TEXTLIST S1_Alarms
  0 = 'Station 1 Clamp A1 Failed to Advance... Check Q1.0...' | German: 'S1 0 Row 1 Failed To Advance.. Check Qxxx.x German' | French: 'S1 0 Row 1 Failed To Advance.. Check Qxxx.x French' | 汉语: '汉语'
  1 = 'Station 1 Clamp A1 Failed to Return... Check Q1.1...' | German: 'S1 1 Row 1 Failed To Return.. Check Qxxx.x German' | French: 'S1 1 Row 1 Failed To Return.. Check Qxxx.x French' | 汉语: '汉语'
  2 = 'Station 1 Clamp A1 Lost Advanced... Check I1.0...' | German: 'S1 2 Row 1 Lost Advance Position... Check Ixxx.x German' | French: 'S1 2 Row 1 Lost Advance Position... Check Ixxx.x French' | 汉语: '汉语'
  3 = 'Station 1 Clamp A1 Lost Returned... Check I1.1...' | German: 'S1 3 Row 1 Lost Return Position... Check Ixxx.x German' | French: 'S1 3 Row 1 Lost Return Position... Check Ixxx.x French'
  4 = 'Station 1 Clamp A1 Switch Fault... Check I1.0, I1.1...' | German: 'S1 4 Row 1 Switch Fault... Check Ixxx.x / Ixxx.x German' | French: 'S1 4 Row 1 Switch Fault... Check Ixxx.x / Ixxx.x French'
  5 = 'Spare' | German: 'S1 5 Row 1 Spare Message German' | French: 'S1 5 Row 1 Spare Message French'
  6 = 'Spare' | German: 'S1 6 Row 1 Spare Message German' | French: 'S1 6 Row 1 Spare Message French'
  7 = 'Spare' | German: 'S1 7 Row 1 Spare Message German' | French: 'S1 7 Row 1 Spare Message French'
  8 = 'Spare' | German: 'S1 8 Row 1 Spare Message German' | French: 'S1 8 Row 1 Spare Message French'
  9 = 'Spare' | German: 'S1 9 Row 1 Spare Message German' | French: 'S1 9 Row 1 Spare Message French'
  10 = 'Lock Cylinder A2 Failed to Lock... Check Q1.2...' | German: 'S1 10 Row 2 Failed To Advance.. Check Qxxx.x German' | French: 'S1 10 Row 2 Failed To Advance.. Check Qxxx.x French'
  11 = 'Lock Cylinder A2 Failed to Unlock... Check Q1.3...' | German: 'S1 11 Row 2 Failed To Return.. Check Qxxx.x German' | French: 'S1 11 Row 2 Failed To Return.. Check Qxxx.x French'
  12 = 'Lock Cylinder A2 Lost Locked... Check I1.2...' | German: 'S1 12 Row 2 Lost Advance Position... Check Ixxx.x German' | French: 'S1 12 Row 2 Lost Advance Position... Check Ixxx.x French'
  13 = 'Lock Cylinder A2 Lost Unlocked... Check I1.3...' | German: 'S1 13 Row 2 Lost Return Position... Check Ixxx.x German' | French: 'S1 13 Row 2 Lost Return Position... Check Ixxx.x French'
  14 = 'Lock Cylinder A2 Switch Fault... Check I1.2, I1.3...' | German: 'S1 14 Row 2 Switch Fault... Check Ixxx.x / Ixxx.x German' | French: 'S1 14 Row 2 Switch Fault... Check Ixxx.x / Ixxx.x French'
  15 = 'Spare' | German: 'S1 15 Row 2 Spare Message German' | French: 'S1 15 Row 2 Spare Message French'
  16 = 'Spare' | German: 'S1 16 Row 2 Spare Message German' | French: 'S1 16 Row 2 Spare Message French'
  17 = 'Spare' | German: 'S1 17 Row 2 Spare Message German' | French: 'S1 17 Row 2 Spare Message French'
  18 = 'Spare' | German: 'S1 18 Row 2 Spare Message German' | French: 'S1 18 Row 2 Spare Message French'
  19 = 'Spare' | German: 'S1 19 Row 2 Spare Message German' | French: 'S1 19 Row 2 Spare Message French'
  20 = 'Urger Cylinder A3 Failed to Urge... Check Q1.4...' | German: 'S1 20 Row 3 Failed To Advance.. Check Qxxx.x German' | French: 'S1 20 Row 3 Failed To Advance.. Check Qxxx.x French'
  21 = 'Urger Cylinder A3 Failed to Return... Check Q1.5...' | German: 'S1 21 Row 3 Failed To Return.. Check Qxxx.x German' | French: 'S1 21 Row 3 Failed To Return.. Check Qxxx.x French'
  22 = 'Urger Cylinder A3 Lost Urged... Check I1.4...' | German: 'S1 22 Row 3 Lost Advance Position... Check Ixxx.x German' | French: 'S1 22 Row 3 Lost Advance Position... Check Ixxx.x French'
  23 = 'Urger Cylinder A3 Lost Returned... Check I1.5...' | German: 'S1 23 Row 3 Lost Return Position... Check Ixxx.x German' | French: 'S1 23 Row 3 Lost Return Position... Check Ixxx.x French'
  24 = 'Urger Cylinder A3 Switch Fault... Check I1.4, I1.5...' | German: 'S1 24 Row 3 Switch Fault... Check Ixxx.x / Ixxx.x German' | French: 'S1 24 Row 3 Switch Fault... Check Ixxx.x / Ixxx.x French'
  25 = 'Spare' | German: 'S1 25 Row 3 Spare Message German' | French: 'S1 25 Row 3 Spare Message French'
  26 = 'Spare' | German: 'S1 26 Row 3 Spare Message German' | French: 'S1 26 Row 3 Spare Message French'
  27 = 'Spare' | German: 'S1 27 Row 3 Spare Message German' | French: 'S1 27 Row 3 Spare Message French'
  28 = 'Spare' | German: 'S1 28 Row 3 Spare Message German' | French: 'S1 28 Row 3 Spare Message French'
  29 = 'Spare' | German: 'S1 29 Row 3 Spare Message German' | French: 'S1 29 Row 3 Spare Message French'
  30 = 'Clamp Cylinder A1 Failed to Advance... Check Q1.0...' | German: 'S1 30 Row 4 Failed To Advance.. Check Qxxx.x German' | French: 'S1 30 Row 4 Failed To Advance.. Check Qxxx.x French'
  31 = 'Clamp Cylinder A1 Failed to Return... Check Q1.1...' | German: 'S1 31 Row 4 Failed To Return.. Check Qxxx.x German' | French: 'S1 31 Row 4 Failed To Return.. Check Qxxx.x French'
  32 = 'Clamp Cylinder A1 Lost Advanced... Check I1.0...' | German: 'S1 32 Row 4 Lost Advance Position... Check Ixxx.x German' | French: 'S1 32 Row 4 Lost Advance Position... Check Ixxx.x French'
  33 = 'Clamp Cylinder A1 Lost Returned... Check I1.1...' | German: 'S1 33 Row 4 Lost Return Position... Check Ixxx.x German' | French: 'S1 33 Row 4 Lost Return Position... Check Ixxx.x French'
  34 = 'Clamp Cylinder A1 Switch Fault... Check I1.0, I1.1...' | German: 'S1 34 Row 4 Switch Fault... Check Ixxx.x / Ixxx.x German' | French: 'S1 34 Row 4 Switch Fault... Check Ixxx.x / Ixxx.x French'
  35 = 'Spare' | German: 'S1 35 Row 4 Spare Message German' | French: 'S1 35 Row 4 Spare Message French'
  36 = 'Spare' | German: 'S1 36 Row 4 Spare Message German' | French: 'S1 36 Row 4 Spare Message French'
  37 = 'Spare' | German: 'S1 37 Row 4 Spare Message German' | French: 'S1 37 Row 4 Spare Message French'
  38 = 'Spare' | German: 'S1 38 Row 4 Spare Message German' | French: 'S1 38 Row 4 Spare Message French'
  39 = 'Spare' | German: 'S1 39 Row 4 Spare Message German' | French: 'S1 39 Row 4 Spare Message French'
  40 = 'Clamp Cylinder A1 Failed to Advance... Check Q1.0...' | German: 'S1 40 Row 5 Failed To Advance.. Check Qxxx.x German' | French: 'S1 40 Row 5 Failed To Advance.. Check Qxxx.x French'
  41 = 'Clamp Cylinder A1 Failed to Return... Check Q1.1...' | German: 'S1 41 Row 5 Failed To Return.. Check Qxxx.x German' | French: 'S1 41 Row 5 Failed To Return.. Check Qxxx.x French'
  42 = 'Clamp Cylinder A1 Lost Advanced... Check I1.0...' | German: 'S1 42 Row 5 Lost Advance Position... Check Ixxx.x German' | French: 'S1 42 Row 5 Lost Advance Position... Check Ixxx.x French'
  43 = 'Clamp Cylinder A1 Lost Returned... Check I1.1...' | German: 'S1 43 Row 5 Lost Return Position... Check Ixxx.x German' | French: 'S1 43 Row 5 Lost Return Position... Check Ixxx.x French'
  44 = 'Clamp Cylinder A1 Switch Fault... Check I1.0, I1.1...' | German: 'S1 44 Row 5 Switch Fault... Check Ixxx.x / Ixxx.x German' | French: 'S1 44 Row 5 Switch Fault... Check Ixxx.x / Ixxx.x French'
  45 = 'Spare' | German: 'S1 45 Row 5 Spare Message German' | French: 'S1 45 Row 5 Spare Message French'
  46 = 'Spare' | German: 'S1 46 Row 5 Spare Message German' | French: 'S1 46 Row 5 Spare Message French'
  47 = 'Spare' | German: 'S1 47 Row 5 Spare Message German' | French: 'S1 47 Row 5 Spare Message French'
  48 = 'Spare' | German: 'S1 48 Row 5 Spare Message German' | French: 'S1 48 Row 5 Spare Message French'
  49 = 'Spare' | German: 'S1 49 Row 5 Spare Message German' | French: 'S1 49 Row 5 Spare Message French'
  50 = 'Clamp Cylinder A1 Failed to Advance... Check Q1.0...' | German: 'S1 50 Row 6 Failed To Advance.. Check Qxxx.x German' | French: 'S1 50 Row 6 Failed To Advance.. Check Qxxx.x French'
  51 = 'Clamp Cylinder A1 Failed to Return... Check Q1.1...' | German: 'S1 51 Row 6 Failed To Return.. Check Qxxx.x German' | French: 'S1 51 Row 6 Failed To Return.. Check Qxxx.x French'
  52 = 'Clamp Cylinder A1 Lost Advanced... Check I1.0...' | German: 'S1 52 Row 6 Lost Advance Position... Check Ixxx.x German' | French: 'S1 52 Row 6 Lost Advance Position... Check Ixxx.x French'
  53 = 'Clamp Cylinder A1 Lost Returned... Check I1.1...' | German: 'S1 53 Row 6 Lost Return Position... Check Ixxx.x German' | French: 'S1 53 Row 6 Lost Return Position... Check Ixxx.x French'
  54 = 'Clamp Cylinder A1 Switch Fault... Check I1.0, I1.1...' | German: 'S1 54 Row 6 Switch Fault... Check Ixxx.x / Ixxx.x German' | French: 'S1 54 Row 6 Switch Fault... Check Ixxx.x / Ixxx.x French'
  55 = 'Spare' | German: 'S1 55 Row 6 Spare Message German' | French: 'S1 55 Row 6 Spare Message French'
  56 = 'Spare' | German: 'S1 56 Row 6 Spare Message German' | French: 'S1 56 Row 6 Spare Message French'
  57 = 'Spare' | German: 'S1 57 Row 6 Spare Message German' | French: 'S1 57 Row 6 Spare Message French'
  58 = 'Spare' | German: 'S1 58 Row 6 Spare Message German' | French: 'S1 58 Row 6 Spare Message French'
  59 = 'Spare' | German: 'S1 59 Row 6 Spare Message German' | French: 'S1 59 Row 6 Spare Message French'
  60 = 'Clamp Cylinder A1 Failed to Advance... Check Q1.0...' | German: 'S1 60 Row 7 Failed To Advance.. Check Qxxx.x German' | French: 'S1 60 Row 7 Failed To Advance.. Check Qxxx.x French'
  61 = 'Clamp Cylinder A1 Failed to Return... Check Q1.1...' | German: 'S1 61 Row 7 Failed To Return.. Check Qxxx.x German' | French: 'S1 61 Row 7 Failed To Return.. Check Qxxx.x French'
  62 = 'Clamp Cylinder A1 Lost Advanced... Check I1.0...' | German: 'S1 62 Row 7 Lost Advance Position... Check Ixxx.x German' | French: 'S1 62 Row 7 Lost Advance Position... Check Ixxx.x French'
  63 = 'Clamp Cylinder A1 Lost Returned... Check I1.1...' | German: 'S1 63 Row 7 Lost Return Position... Check Ixxx.x German' | French: 'S1 63 Row 7 Lost Return Position... Check Ixxx.x French'
  64 = 'Clamp Cylinder A1 Switch Fault... Check I1.0, I1.1...' | German: 'S1 64 Row 7 Switch Fault... Check Ixxx.x / Ixxx.x German' | French: 'S1 64 Row 7 Switch Fault... Check Ixxx.x / Ixxx.x French'
  65 = 'Spare' | German: 'S1 65 Row 7 Spare Message German' | French: 'S1 65 Row 7 Spare Message French'
  66 = 'Spare' | German: 'S1 66 Row 7 Spare Message German' | French: 'S1 66 Row 7 Spare Message French'
  67 = 'Spare' | German: 'S1 67 Row 7 Spare Message German' | French: 'S1 67 Row 7 Spare Message French'
  68 = 'Spare' | German: 'S1 68 Row 7 Spare Message German' | French: 'S1 68 Row 7 Spare Message French'
  69 = 'Spare' | German: 'S1 69 Row 7 Spare Message German' | French: 'S1 69 Row 7 Spare Message French'
  70 = 'Clamp Cylinder A1 Failed to Advance... Check Q1.0...' | German: 'S1 70 Row 8 Failed To Advance.. Check Qxxx.x German' | French: 'S1 70 Row 8 Failed To Advance.. Check Qxxx.x French'
  71 = 'Clamp Cylinder A1 Failed to Return... Check Q1.1...' | German: 'S1 71 Row 8 Failed To Return.. Check Qxxx.x German' | French: 'S1 71 Row 8 Failed To Return.. Check Qxxx.x French'
  72 = 'Clamp Cylinder A1 Lost Advanced... Check I1.0...' | German: 'S1 72 Row 8 Lost Advance Position... Check Ixxx.x German' | French: 'S1 72 Row 8 Lost Advance Position... Check Ixxx.x French'
  73 = 'Clamp Cylinder A1 Lost Returned... Check I1.1...' | German: 'S1 73 Row 8 Lost Return Position... Check Ixxx.x German' | French: 'S1 73 Row 8 Lost Return Position... Check Ixxx.x French'
  74 = 'Clamp Cylinder A1 Switch Fault... Check I1.0, I1.1...' | German: 'S1 74 Row 8 Switch Fault... Check Ixxx.x / Ixxx.x German' | French: 'S1 74 Row 8 Switch Fault... Check Ixxx.x / Ixxx.x French'
  75 = 'Spare' | German: 'S1 75 Row 8 Spare Message German' | French: 'S1 75 Row 8 Spare Message French'
  76 = 'Spare' | German: 'S1 76 Row 8 Spare Message German' | French: 'S1 76 Row 8 Spare Message French'
  77 = 'Spare' | German: 'S1 77 Row 8 Spare Message German' | French: 'S1 77 Row 8 Spare Message French'
  78 = 'Spare' | German: 'S1 78 Row 8 Spare Message German' | French: 'S1 78 Row 8 Spare Message French'
  79 = 'Spare' | German: 'S1 79 Row 8 Spare Message German' | French: 'S1 79 Row 8 Spare Message French'
  80 = 'Clamp Cylinder A1 Failed to Advance... Check Q1.0...' | German: 'S1 80 Row 9 Failed To Advance.. Check Qxxx.x German' | French: 'S1 80 Row 9 Failed To Advance.. Check Qxxx.x French'
  81 = 'Clamp Cylinder A1 Failed to Return... Check Q1.1...' | German: 'S1 81 Row 9 Failed To Return.. Check Qxxx.x German' | French: 'S1 81 Row 9 Failed To Return.. Check Qxxx.x French'
  82 = 'Clamp Cylinder A1 Lost Advanced... Check I1.0...' | German: 'S1 82 Row 9 Lost Advance Position... Check Ixxx.x German' | French: 'S1 82 Row 9 Lost Advance Position... Check Ixxx.x French'
  83 = 'Clamp Cylinder A1 Lost Returned... Check I1.1...' | German: 'S1 83 Row 9 Lost Return Position... Check Ixxx.x German' | French: 'S1 83 Row 9 Lost Return Position... Check Ixxx.x French'
  84 = 'Clamp Cylinder A1 Switch Fault... Check I1.0, I1.1...' | German: 'S1 84 Row 9 Switch Fault... Check Ixxx.x / Ixxx.x German' | French: 'S1 84 Row 9 Switch Fault... Check Ixxx.x / Ixxx.x French'
  85 = 'Spare' | German: 'S1 85 Row 9 Spare Message German' | French: 'S1 85 Row 9 Spare Message French'
  86 = 'Spare' | German: 'S1 86 Row 9 Spare Message German' | French: 'S1 86 Row 9 Spare Message French'
  87 = 'Spare' | German: 'S1 87 Row 9 Spare Message German' | French: 'S1 87 Row 9 Spare Message French'
  88 = 'Spare' | German: 'S1 88 Row 9 Spare Message German' | French: 'S1 88 Row 9 Spare Message French'
  89 = 'Spare' | German: 'S1 89 Row 9 Spare Message German' | French: 'S1 89 Row 9 Spare Message French'
  90 = 'Clamp Cylinder A1 Failed to Advance... Check Q1.0...' | German: 'S1 90 Row 10 Failed To Advance.. Check Qxxx.x German' | French: 'S1 90 Row 10 Failed To Advance.. Check Qxxx.x French'
  91 = 'Clamp Cylinder A1 Failed to Return... Check Q1.1...' | German: 'S1 91 Row 10 Failed To Return.. Check Qxxx.x German' | French: 'S1 91 Row 10 Failed To Return.. Check Qxxx.x French'
  92 = 'Clamp Cylinder A1 Lost Advanced... Check I1.0...' | German: 'S1 92 Row 10 Lost Advance Position... Check Ixxx.x German' | French: 'S1 92 Row 10 Lost Advance Position... Check Ixxx.x French'
  93 = 'Clamp Cylinder A1 Lost Returned... Check I1.1...' | German: 'S1 93 Row 10 Lost Return Position... Check Ixxx.x German' | French: 'S1 93 Row 10 Lost Return Position... Check Ixxx.x French'
  94 = 'Clamp Cylinder A1 Switch Fault... Check I1.0, I1.1...' | German: 'S1 94 Row 10 Switch Fault... Check Ixxx.x / Ixxx.x German' | French: 'S1 94 Row 10 Switch Fault... Check Ixxx.x / Ixxx.x French'
  95 = 'Spare' | German: 'S1 95 Row 10 Spare Message German' | French: 'S1 95 Row 10 Spare Message French'
  96 = 'Spare' | German: 'S1 96 Row 10 Spare Message German' | French: 'S1 96 Row 10 Spare Message French'
  97 = 'Spare' | German: 'S1 97 Row 10 Spare Message German' | French: 'S1 97 Row 10 Spare Message French'
  98 = 'Spare' | German: 'S1 98 Row 10 Spare Message German' | French: 'S1 98 Row 10 Spare Message French'
  99 = 'Spare' | German: 'S1 99 Row 10 Spare Message German' | French: 'S1 99 Row 10 Spare Message French'
  100 = 'Clamp Cylinder A1 Failed to Advance... Check Q1.0...' | German: 'S1 100 Row 11 Failed To Advance.. Check Qxxx.x German' | French: 'S1 100 Row 11 Failed To Advance.. Check Qxxx.x French'
  101 = 'Clamp Cylinder A1 Failed to Return... Check Q1.1...' | German: 'S1 101 Row 11 Failed To Return.. Check Qxxx.x German' | French: 'S1 101 Row 11 Failed To Return.. Check Qxxx.x French'
  102 = 'Clamp Cylinder A1 Lost Advanced... Check I1.0...' | German: 'S1 102 Row 11 Lost Advance Position... Check Ixxx.x German' | French: 'S1 102 Row 11 Lost Advance Position... Check Ixxx.x French'
  103 = 'Clamp Cylinder A1 Lost Returned... Check I1.1...' | German: 'S1 103 Row 11 Lost Return Position... Check Ixxx.x German' | French: 'S1 103 Row 11 Lost Return Position... Check Ixxx.x French'
  104 = 'Clamp Cylinder A1 Switch Fault... Check I1.0, I1.1...' | German: 'S1 104 Row 11 Switch Fault... Check Ixxx.x / Ixxx.x German' | French: 'S1 104 Row 11 Switch Fault... Check Ixxx.x / Ixxx.x French'
  105 = 'Spare' | German: 'S1 105 Row 11 Spare Message German' | French: 'S1 105 Row 11 Spare Message French'
  106 = 'Spare' | German: 'S1 106 Row 11 Spare Message German' | French: 'S1 106 Row 11 Spare Message French'
  107 = 'Spare' | German: 'S1 107 Row 11 Spare Message German' | French: 'S1 107 Row 11 Spare Message French'
  108 = 'Spare' | German: 'S1 108 Row 11 Spare Message German' | French: 'S1 108 Row 11 Spare Message French'
  109 = 'Spare' | German: 'S1 109 Row 11 Spare Message German' | French: 'S1 109 Row 11 Spare Message French'
  110 = 'Clamp Cylinder A1 Failed to Advance... Check Q1.0...' | German: 'S1 110 Row 12 Failed To Advance.. Check Qxxx.x German' | French: 'S1 110 Row 12 Failed To Advance.. Check Qxxx.x French'
  111 = 'Clamp Cylinder A1 Failed to Return... Check Q1.1...' | German: 'S1 111 Row 12 Failed To Return.. Check Qxxx.x German' | French: 'S1 111 Row 12 Failed To Return.. Check Qxxx.x French'
  112 = 'Clamp Cylinder A1 Lost Advanced... Check I1.0...' | German: 'S1 112 Row 12 Lost Advance Position... Check Ixxx.x German' | French: 'S1 112 Row 12 Lost Advance Position... Check Ixxx.x French'
  113 = 'Clamp Cylinder A1 Lost Returned... Check I1.1...' | German: 'S1 113 Row 12 Lost Return Position... Check Ixxx.x German' | French: 'S1 113 Row 12 Lost Return Position... Check Ixxx.x French'
  114 = 'Clamp Cylinder A1 Switch Fault... Check I1.0, I1.1...' | German: 'S1 114 Row 12 Switch Fault... Check Ixxx.x / Ixxx.x German' | French: 'S1 114 Row 12 Switch Fault... Check Ixxx.x / Ixxx.x French'
  115 = 'Spare' | German: 'S1 115 Row 12 Spare Message German' | French: 'S1 115 Row 12 Spare Message French'
  116 = 'Spare' | German: 'S1 116 Row 12 Spare Message German' | French: 'S1 116 Row 12 Spare Message French'
  117 = 'Spare' | German: 'S1 117 Row 12 Spare Message German' | French: 'S1 117 Row 12 Spare Message French'
  118 = 'Spare' | German: 'S1 118 Row 12 Spare Message German' | French: 'S1 118 Row 12 Spare Message French'
  119 = 'Spare' | German: 'S1 119 Row 12 Spare Message German' | French: 'S1 119 Row 12 Spare Message French'
  120 = 'Clamp Cylinder A1 Failed to Advance... Check Q1.0...' | German: 'S1 120 Row 13 Failed To Advance.. Check Qxxx.x German' | French: 'S1 120 Row 13 Failed To Advance.. Check Qxxx.x French'
  121 = 'Clamp Cylinder A1 Failed to Return... Check Q1.1...' | German: 'S1 121 Row 13 Failed To Return.. Check Qxxx.x German' | French: 'S1 121 Row 13 Failed To Return.. Check Qxxx.x French'
  122 = 'Clamp Cylinder A1 Lost Advanced... Check I1.0...' | German: 'S1 122 Row 13 Lost Advance Position... Check Ixxx.x German' | French: 'S1 122 Row 13 Lost Advance Position... Check Ixxx.x French'
  123 = 'Clamp Cylinder A1 Lost Returned... Check I1.1...' | German: 'S1 123 Row 13 Lost Return Position... Check Ixxx.x German' | French: 'S1 123 Row 13 Lost Return Position... Check Ixxx.x French'
  124 = 'Clamp Cylinder A1 Switch Fault... Check I1.0, I1.1...' | German: 'S1 124 Row 13 Switch Fault... Check Ixxx.x / Ixxx.x German' | French: 'S1 124 Row 13 Switch Fault... Check Ixxx.x / Ixxx.x French'
  125 = 'Spare' | German: 'S1 125 Row 13 Spare Message German' | French: 'S1 125 Row 13 Spare Message French'
  126 = 'Spare' | German: 'S1 126 Row 13 Spare Message German' | French: 'S1 126 Row 13 Spare Message French'
  127 = 'Spare' | German: 'S1 127 Row 13 Spare Message German' | French: 'S1 127 Row 13 Spare Message French'
  128 = 'Spare' | German: 'S1 128 Row 13 Spare Message German' | French: 'S1 128 Row 13 Spare Message French'
  129 = 'Spare' | German: 'S1 129 Row 13 Spare Message German' | French: 'S1 129 Row 13 Spare Message French'
  130 = 'Clamp Cylinder A1 Failed to Advance... Check Q1.0...' | German: 'S1 130 Row 14 Failed To Advance.. Check Qxxx.x German' | French: 'S1 130 Row 14 Failed To Advance.. Check Qxxx.x French'
  131 = 'Clamp Cylinder A1 Failed to Return... Check Q1.1...' | German: 'S1 131 Row 14 Failed To Return.. Check Qxxx.x German' | French: 'S1 131 Row 14 Failed To Return.. Check Qxxx.x French'
  132 = 'Clamp Cylinder A1 Lost Advanced... Check I1.0...' | German: 'S1 132 Row 14 Lost Advance Position... Check Ixxx.x German' | French: 'S1 132 Row 14 Lost Advance Position... Check Ixxx.x French'
  133 = 'Clamp Cylinder A1 Lost Returned... Check I1.1...' | German: 'S1 133 Row 14 Lost Return Position... Check Ixxx.x German' | French: 'S1 133 Row 14 Lost Return Position... Check Ixxx.x French'
  134 = 'Clamp Cylinder A1 Switch Fault... Check I1.0, I1.1...' | German: 'S1 134 Row 14 Switch Fault... Check Ixxx.x / Ixxx.x German' | French: 'S1 134 Row 14 Switch Fault... Check Ixxx.x / Ixxx.x French'
  135 = 'Spare' | German: 'S1 135 Row 14 Spare Message German' | French: 'S1 135 Row 14 Spare Message French'
  136 = 'Spare' | German: 'S1 136 Row 14 Spare Message German' | French: 'S1 136 Row 14 Spare Message French'
  137 = 'Spare' | German: 'S1 137 Row 14 Spare Message German' | French: 'S1 137 Row 14 Spare Message French'
  138 = 'Spare' | German: 'S1 138 Row 14 Spare Message German' | French: 'S1 138 Row 14 Spare Message French'
  139 = 'Spare' | German: 'S1 139 Row 14 Spare Message German' | French: 'S1 139 Row 14 Spare Message French'
  140 = 'Clamp Cylinder A1 Failed to Advance... Check Q1.0...' | German: 'S1 140 Row 15 Failed To Advance.. Check Qxxx.x German' | French: 'S1 140 Row 15 Failed To Advance.. Check Qxxx.x French'
  141 = 'Clamp Cylinder A1 Failed to Return... Check Q1.1...' | German: 'S1 141 Row 15 Failed To Return.. Check Qxxx.x German' | French: 'S1 141 Row 15 Failed To Return.. Check Qxxx.x French'
  142 = 'Clamp Cylinder A1 Lost Advanced... Check I1.0...' | German: 'S1 142 Row 15 Lost Advance Position... Check Ixxx.x German' | French: 'S1 142 Row 15 Lost Advance Position... Check Ixxx.x French'
  143 = 'Clamp Cylinder A1 Lost Returned... Check I1.1...' | German: 'S1 143 Row 15 Lost Return Position... Check Ixxx.x German' | French: 'S1 143 Row 15 Lost Return Position... Check Ixxx.x French'
  144 = 'Clamp Cylinder A1 Switch Fault... Check I1.0, I1.1...' | German: 'S1 144 Row 15 Switch Fault... Check Ixxx.x / Ixxx.x German' | French: 'S1 144 Row 15 Switch Fault... Check Ixxx.x / Ixxx.x French'
  145 = 'Spare' | German: 'S1 145 Row 15 Spare Message German' | French: 'S1 145 Row 15 Spare Message French'
  146 = 'Spare' | German: 'S1 146 Row 15 Spare Message German' | French: 'S1 146 Row 15 Spare Message French'
  147 = 'Spare' | German: 'S1 147 Row 15 Spare Message German' | French: 'S1 147 Row 15 Spare Message French'
  148 = 'Spare' | German: 'S1 148 Row 15 Spare Message German' | French: 'S1 148 Row 15 Spare Message French'
  149 = 'Spare' | German: 'S1 149 Row 15 Spare Message German' | French: 'S1 149 Row 15 Spare Message French'
  150 = 'Clamp Cylinder A1 Failed to Advance... Check Q1.0...' | German: 'S1 150 Row 16 Failed To Advance.. Check Qxxx.x German' | French: 'S1 150 Row 16 Failed To Advance.. Check Qxxx.x French'
  151 = 'Clamp Cylinder A1 Failed to Return... Check Q1.1...' | German: 'S1 151 Row 16 Failed To Return.. Check Qxxx.x German' | French: 'S1 151 Row 16 Failed To Return.. Check Qxxx.x French'
  152 = 'Clamp Cylinder A1 Lost Advanced... Check I1.0...' | German: 'S1 152 Row 16 Lost Advance Position... Check Ixxx.x German' | French: 'S1 152 Row 16 Lost Advance Position... Check Ixxx.x French'
  153 = 'Clamp Cylinder A1 Lost Returned... Check I1.1...' | German: 'S1 153 Row 16 Lost Return Position... Check Ixxx.x German' | French: 'S1 153 Row 16 Lost Return Position... Check Ixxx.x French'
  154 = 'Clamp Cylinder A1 Switch Fault... Check I1.0, I1.1...' | German: 'S1 154 Row 16 Switch Fault... Check Ixxx.x / Ixxx.x German' | French: 'S1 154 Row 16 Switch Fault... Check Ixxx.x / Ixxx.x French'
  155 = 'Spare' | German: 'S1 155 Row 16 Spare Message German' | French: 'S1 155 Row 16 Spare Message French'
  156 = 'Spare' | German: 'S1 156 Row 16 Spare Message German' | French: 'S1 156 Row 16 Spare Message French'
  157 = 'Spare' | German: 'S1 157 Row 16 Spare Message German' | French: 'S1 157 Row 16 Spare Message French'
  158 = 'Spare' | German: 'S1 158 Row 16 Spare Message German' | French: 'S1 158 Row 16 Spare Message French'
  159 = 'Spare' | German: 'S1 159 Row 16 Spare Message German' | French: 'S1 159 Row 16 Spare Message French'
  160 = 'Clamp Cylinder A1 Failed to Advance... Check Q1.0...' | German: 'S1 160 Row 17 Failed To Advance.. Check Qxxx.x German' | French: 'S1 160 Row 17 Failed To Advance.. Check Qxxx.x French'
  161 = 'Clamp Cylinder A1 Failed to Return... Check Q1.1...' | German: 'S1 161 Row 17 Failed To Return.. Check Qxxx.x German' | French: 'S1 161 Row 17 Failed To Return.. Check Qxxx.x French'
  162 = 'Clamp Cylinder A1 Lost Advanced... Check I1.0...' | German: 'S1 162 Row 17 Lost Advance Position... Check Ixxx.x German' | French: 'S1 162 Row 17 Lost Advance Position... Check Ixxx.x French'
  163 = 'Clamp Cylinder A1 Lost Returned... Check I1.1...' | German: 'S1 163 Row 17 Lost Return Position... Check Ixxx.x German' | French: 'S1 163 Row 17 Lost Return Position... Check Ixxx.x French'
  164 = 'Clamp Cylinder A1 Switch Fault... Check I1.0, I1.1...' | German: 'S1 164 Row 17 Switch Fault... Check Ixxx.x / Ixxx.x German' | French: 'S1 164 Row 17 Switch Fault... Check Ixxx.x / Ixxx.x French'
  165 = 'Spare' | German: 'S1 165 Row 17 Spare Message German' | French: 'S1 165 Row 17 Spare Message French'
  166 = 'Spare' | German: 'S1 166 Row 17 Spare Message German' | French: 'S1 166 Row 17 Spare Message French'
  167 = 'Spare' | German: 'S1 167 Row 17 Spare Message German' | French: 'S1 167 Row 17 Spare Message French'
  168 = 'Spare' | German: 'S1 168 Row 17 Spare Message German' | French: 'S1 168 Row 17 Spare Message French'
  169 = 'Spare' | German: 'S1 169 Row 17 Spare Message German' | French: 'S1 169 Row 17 Spare Message French'
  170 = 'Clamp Cylinder A1 Failed to Advance... Check Q1.0...' | German: 'S1 170 Row 18 Failed To Advance.. Check Qxxx.x German' | French: 'S1 170 Row 18 Failed To Advance.. Check Qxxx.x French'
  171 = 'Clamp Cylinder A1 Failed to Return... Check Q1.1...' | German: 'S1 171 Row 18 Failed To Return.. Check Qxxx.x German' | French: 'S1 171 Row 18 Failed To Return.. Check Qxxx.x French'
  172 = 'Clamp Cylinder A1 Lost Advanced... Check I1.0...' | German: 'S1 172 Row 18 Lost Advance Position... Check Ixxx.x German' | French: 'S1 172 Row 18 Lost Advance Position... Check Ixxx.x French'
  173 = 'Clamp Cylinder A1 Lost Returned... Check I1.1...' | German: 'S1 173 Row 18 Lost Return Position... Check Ixxx.x German' | French: 'S1 173 Row 18 Lost Return Position... Check Ixxx.x French'
  174 = 'Clamp Cylinder A1 Switch Fault... Check I1.0, I1.1...' | German: 'S1 174 Row 18 Switch Fault... Check Ixxx.x / Ixxx.x German' | French: 'S1 174 Row 18 Switch Fault... Check Ixxx.x / Ixxx.x French'
  175 = 'Spare' | German: 'S1 175 Row 18 Spare Message German' | French: 'S1 175 Row 18 Spare Message French'
  176 = 'Spare' | German: 'S1 176 Row 18 Spare Message German' | French: 'S1 176 Row 18 Spare Message French'
  177 = 'Spare' | German: 'S1 177 Row 18 Spare Message German' | French: 'S1 177 Row 18 Spare Message French'
  178 = 'Spare' | German: 'S1 178 Row 18 Spare Message German' | French: 'S1 178 Row 18 Spare Message French'
  179 = 'Spare' | German: 'S1 179 Row 18 Spare Message German' | French: 'S1 179 Row 18 Spare Message French'
  180 = 'Clamp Cylinder A1 Failed to Advance... Check Q1.0...' | German: 'S1 180 Row 19 Failed To Advance.. Check Qxxx.x German' | French: 'S1 180 Row 19 Failed To Advance.. Check Qxxx.x French'
  181 = 'Clamp Cylinder A1 Failed to Return... Check Q1.1...' | German: 'S1 181 Row 19 Failed To Return.. Check Qxxx.x German' | French: 'S1 181 Row 19 Failed To Return.. Check Qxxx.x French'
  182 = 'Clamp Cylinder A1 Lost Advanced... Check I1.0...' | German: 'S1 182 Row 19 Lost Advance Position... Check Ixxx.x German' | French: 'S1 182 Row 19 Lost Advance Position... Check Ixxx.x French'
  183 = 'Clamp Cylinder A1 Lost Returned... Check I1.1...' | German: 'S1 183 Row 19 Lost Return Position... Check Ixxx.x German' | French: 'S1 183 Row 19 Lost Return Position... Check Ixxx.x French'
  184 = 'Clamp Cylinder A1 Switch Fault... Check I1.0, I1.1...' | German: 'S1 184 Row 19 Switch Fault... Check Ixxx.x / Ixxx.x German' | French: 'S1 184 Row 19 Switch Fault... Check Ixxx.x / Ixxx.x French'
  185 = 'Spare' | German: 'S1 185 Row 19 Spare Message German' | French: 'S1 185 Row 19 Spare Message French'
  186 = 'Spare' | German: 'S1 186 Row 19 Spare Message German' | French: 'S1 186 Row 19 Spare Message French'
  187 = 'Spare' | German: 'S1 187 Row 19 Spare Message German' | French: 'S1 187 Row 19 Spare Message French'
  188 = 'Spare' | German: 'S1 188 Row 19 Spare Message German' | French: 'S1 188 Row 19 Spare Message French'
  189 = 'Spare' | German: 'S1 189 Row 19 Spare Message German' | French: 'S1 189 Row 19 Spare Message French'
  190 = 'Clamp Cylinder A1 Failed to Advance... Check Q1.0...' | German: 'S1 190 Row 20 Failed To Advance.. Check Qxxx.x German' | French: 'S1 190 Row 20 Failed To Advance.. Check Qxxx.x French'
  191 = 'Clamp Cylinder A1 Failed to Return... Check Q1.1...' | German: 'S1 191 Row 20 Failed To Return.. Check Qxxx.x German' | French: 'S1 191 Row 20 Failed To Return.. Check Qxxx.x French'
  192 = 'Clamp Cylinder A1 Lost Advanced... Check I1.0...' | German: 'S1 192 Row 20 Lost Advance Position... Check Ixxx.x German' | French: 'S1 192 Row 20 Lost Advance Position... Check Ixxx.x French'
  193 = 'Clamp Cylinder A1 Lost Returned... Check I1.1...' | German: 'S1 193 Row 20 Lost Return Position... Check Ixxx.x German' | French: 'S1 193 Row 20 Lost Return Position... Check Ixxx.x French'
  194 = 'Clamp Cylinder A1 Switch Fault... Check I1.0, I1.1...' | German: 'S1 194 Row 20 Switch Fault... Check Ixxx.x / Ixxx.x German' | French: 'S1 194 Row 20 Switch Fault... Check Ixxx.x / Ixxx.x French'
  195 = 'Spare' | German: 'S1 195 Row 20 Spare Message German' | French: 'S1 195 Row 20 Spare Message French'
  196 = 'Spare' | German: 'S1 196 Row 20 Spare Message German' | French: 'S1 196 Row 20 Spare Message French'
  197 = 'Spare' | German: 'S1 197 Row 20 Spare Message German' | French: 'S1 197 Row 20 Spare Message French'
  198 = 'Spare' | German: 'S1 198 Row 20 Spare Message German' | French: 'S1 198 Row 20 Spare Message French'
  199 = 'Spare' | German: 'S1 199 Row 20 Spare Message German' | French: 'S1 199 Row 20 Spare Message French'
  200 = 'Clamp Cylinder A1 Failed to Advance... Check Q1.0...' | German: 'S1 200 Row 21 Failed To Advance.. Check Qxxx.x German' | French: 'S1 200 Row 21 Failed To Advance.. Check Qxxx.x French'
  201 = 'Clamp Cylinder A1 Failed to Return... Check Q1.1...' | German: 'S1 201 Row 21 Failed To Return.. Check Qxxx.x German' | French: 'S1 201 Row 21 Failed To Return.. Check Qxxx.x French'
  202 = 'Clamp Cylinder A1 Lost Advanced... Check I1.0...' | German: 'S1 202 Row 21 Lost Advance Position... Check Ixxx.x German' | French: 'S1 202 Row 21 Lost Advance Position... Check Ixxx.x French'
  203 = 'Clamp Cylinder A1 Lost Returned... Check I1.1...' | German: 'S1 203 Row 21 Lost Return Position... Check Ixxx.x German' | French: 'S1 203 Row 21 Lost Return Position... Check Ixxx.x French'
  204 = 'Clamp Cylinder A1 Switch Fault... Check I1.0, I1.1...' | German: 'S1 204 Row 21 Switch Fault... Check Ixxx.x / Ixxx.x German' | French: 'S1 204 Row 21 Switch Fault... Check Ixxx.x / Ixxx.x French'
  205 = 'Spare' | German: 'S1 205 Row 21 Spare Message German' | French: 'S1 205 Row 21 Spare Message French'
  206 = 'Spare' | German: 'S1 206 Row 21 Spare Message German' | French: 'S1 206 Row 21 Spare Message French'
  207 = 'Spare' | German: 'S1 207 Row 21 Spare Message German' | French: 'S1 207 Row 21 Spare Message French'
  208 = 'Spare' | German: 'S1 208 Row 21 Spare Message German' | French: 'S1 208 Row 21 Spare Message French'
  209 = 'Spare' | German: 'S1 209 Row 21 Spare Message German' | French: 'S1 209 Row 21 Spare Message French'
  210 = 'Clamp Cylinder A1 Failed to Advance... Check Q1.0...' | German: 'S1 210 Row 22 Failed To Advance.. Check Qxxx.x German' | French: 'S1 210 Row 22 Failed To Advance.. Check Qxxx.x French'
  211 = 'Clamp Cylinder A1 Failed to Return... Check Q1.1...' | German: 'S1 211 Row 22 Failed To Return.. Check Qxxx.x German' | French: 'S1 211 Row 22 Failed To Return.. Check Qxxx.x French'
  212 = 'Clamp Cylinder A1 Lost Advanced... Check I1.0...' | German: 'S1 212 Row 22 Lost Advance Position... Check Ixxx.x German' | French: 'S1 212 Row 22 Lost Advance Position... Check Ixxx.x French'
  213 = 'Clamp Cylinder A1 Lost Returned... Check I1.1...' | German: 'S1 213 Row 22 Lost Return Position... Check Ixxx.x German' | French: 'S1 213 Row 22 Lost Return Position... Check Ixxx.x French'
  214 = 'Clamp Cylinder A1 Switch Fault... Check I1.0, I1.1...' | German: 'S1 214 Row 22 Switch Fault... Check Ixxx.x / Ixxx.x German' | French: 'S1 214 Row 22 Switch Fault... Check Ixxx.x / Ixxx.x French'
  215 = 'Spare' | German: 'S1 215 Row 22 Spare Message German' | French: 'S1 215 Row 22 Spare Message French'
  216 = 'Spare' | German: 'S1 216 Row 22 Spare Message German' | French: 'S1 216 Row 22 Spare Message French'
  217 = 'Spare' | German: 'S1 217 Row 22 Spare Message German' | French: 'S1 217 Row 22 Spare Message French'
  218 = 'Spare' | German: 'S1 218 Row 22 Spare Message German' | French: 'S1 218 Row 22 Spare Message French'
  219 = 'Spare' | German: 'S1 219 Row 22 Spare Message German' | French: 'S1 219 Row 22 Spare Message French'
  220 = 'Clamp Cylinder A1 Failed to Advance... Check Q1.0...' | German: 'S1 220 Row 23 Failed To Advance.. Check Qxxx.x German' | French: 'S1 220 Row 23 Failed To Advance.. Check Qxxx.x French'
  221 = 'Clamp Cylinder A1 Failed to Return... Check Q1.1...' | German: 'S1 221 Row 23 Failed To Return.. Check Qxxx.x German' | French: 'S1 221 Row 23 Failed To Return.. Check Qxxx.x French'
  222 = 'Clamp Cylinder A1 Lost Advanced... Check I1.0...' | German: 'S1 222 Row 23 Lost Advance Position... Check Ixxx.x German' | French: 'S1 222 Row 23 Lost Advance Position... Check Ixxx.x French'
  223 = 'Clamp Cylinder A1 Lost Returned... Check I1.1...' | German: 'S1 223 Row 23 Lost Return Position... Check Ixxx.x German' | French: 'S1 223 Row 23 Lost Return Position... Check Ixxx.x French'
  224 = 'Clamp Cylinder A1 Switch Fault... Check I1.0, I1.1...' | German: 'S1 224 Row 23 Switch Fault... Check Ixxx.x / Ixxx.x German' | French: 'S1 224 Row 23 Switch Fault... Check Ixxx.x / Ixxx.x French'
  225 = 'Spare' | German: 'S1 225 Row 23 Spare Message German' | French: 'S1 225 Row 23 Spare Message French'
  226 = 'Spare' | German: 'S1 226 Row 23 Spare Message German' | French: 'S1 226 Row 23 Spare Message French'
  227 = 'Spare' | German: 'S1 227 Row 23 Spare Message German' | French: 'S1 227 Row 23 Spare Message French'
  228 = 'Spare' | German: 'S1 228 Row 23 Spare Message German' | French: 'S1 228 Row 23 Spare Message French'
  229 = 'Spare' | German: 'S1 229 Row 23 Spare Message German' | French: 'S1 229 Row 23 Spare Message French'
  230 = 'Clamp Cylinder A1 Failed to Advance... Check Q1.0...' | German: 'S1 230 Row 24 Failed To Advance.. Check Qxxx.x German' | French: 'S1 230 Row 24 Failed To Advance.. Check Qxxx.x French'
  231 = 'Clamp Cylinder A1 Failed to Return... Check Q1.1...' | German: 'S1 231 Row 24 Failed To Return.. Check Qxxx.x German' | French: 'S1 231 Row 24 Failed To Return.. Check Qxxx.x French'
  232 = 'Clamp Cylinder A1 Lost Advanced... Check I1.0...' | German: 'S1 232 Row 24 Lost Advance Position... Check Ixxx.x German' | French: 'S1 232 Row 24 Lost Advance Position... Check Ixxx.x French'
  233 = 'Clamp Cylinder A1 Lost Returned... Check I1.1...' | German: 'S1 233 Row 24 Lost Return Position... Check Ixxx.x German' | French: 'S1 233 Row 24 Lost Return Position... Check Ixxx.x French'
  234 = 'Clamp Cylinder A1 Switch Fault... Check I1.0, I1.1...' | German: 'S1 234 Row 24 Switch Fault... Check Ixxx.x / Ixxx.x German' | French: 'S1 234 Row 24 Switch Fault... Check Ixxx.x / Ixxx.x French'
  235 = 'Spare' | German: 'S1 235 Row 24 Spare Message German' | French: 'S1 235 Row 24 Spare Message French'
  236 = 'Spare' | German: 'S1 236 Row 24 Spare Message German' | French: 'S1 236 Row 24 Spare Message French'
  237 = 'Spare' | German: 'S1 237 Row 24 Spare Message German' | French: 'S1 237 Row 24 Spare Message French'
  238 = 'Spare' | German: 'S1 238 Row 24 Spare Message German' | French: 'S1 238 Row 24 Spare Message French'
  239 = 'Spare' | German: 'S1 239 Row 24 Spare Message German' | French: 'S1 239 Row 24 Spare Message French'
  240 = 'Clamp Cylinder A1 Failed to Advance... Check Q1.0...' | German: 'S1 240 Row 25 Failed To Advance.. Check Qxxx.x German' | French: 'S1 240 Row 25 Failed To Advance.. Check Qxxx.x French'
  241 = 'Clamp Cylinder A1 Failed to Return... Check Q1.1...' | German: 'S1 241 Row 25 Failed To Return.. Check Qxxx.x German' | French: 'S1 241 Row 25 Failed To Return.. Check Qxxx.x French'
  242 = 'Clamp Cylinder A1 Lost Advanced... Check I1.0...' | German: 'S1 242 Row 25 Lost Advance Position... Check Ixxx.x German' | French: 'S1 242 Row 25 Lost Advance Position... Check Ixxx.x French'
  243 = 'Clamp Cylinder A1 Lost Returned... Check I1.1...' | German: 'S1 243 Row 25 Lost Return Position... Check Ixxx.x German' | French: 'S1 243 Row 25 Lost Return Position... Check Ixxx.x French'
  244 = 'Clamp Cylinder A1 Switch Fault... Check I1.0, I1.1...' | German: 'S1 244 Row 25 Switch Fault... Check Ixxx.x / Ixxx.x German' | French: 'S1 244 Row 25 Switch Fault... Check Ixxx.x / Ixxx.x French'
  245 = 'Spare' | German: 'S1 245 Row 25 Spare Message German' | French: 'S1 245 Row 25 Spare Message French'
  246 = 'Spare' | German: 'S1 246 Row 25 Spare Message German' | French: 'S1 246 Row 25 Spare Message French'
  247 = 'Spare' | German: 'S1 247 Row 25 Spare Message German' | French: 'S1 247 Row 25 Spare Message French'
  248 = 'Spare' | German: 'S1 248 Row 25 Spare Message German' | French: 'S1 248 Row 25 Spare Message French'
  249 = 'Spare' | German: 'S1 249 Row 25 Spare Message German' | French: 'S1 249 Row 25 Spare Message French'
  250 = 'Clamp Cylinder A1 Failed to Advance... Check Q1.0...' | German: 'S1 250 Row 26 Failed To Advance.. Check Qxxx.x German' | French: 'S1 250 Row 26 Failed To Advance.. Check Qxxx.x French'
  251 = 'Clamp Cylinder A1 Failed to Return... Check Q1.1...' | German: 'S1 251 Row 26 Failed To Return.. Check Qxxx.x German' | French: 'S1 251 Row 26 Failed To Return.. Check Qxxx.x French'
  252 = 'Clamp Cylinder A1 Lost Advanced... Check I1.0...' | German: 'S1 252 Row 26 Lost Advance Position... Check Ixxx.x German' | French: 'S1 252 Row 26 Lost Advance Position... Check Ixxx.x French'
  253 = 'Clamp Cylinder A1 Lost Returned... Check I1.1...' | German: 'S1 253 Row 26 Lost Return Position... Check Ixxx.x German' | French: 'S1 253 Row 26 Lost Return Position... Check Ixxx.x French'
  254 = 'Clamp Cylinder A1 Switch Fault... Check I1.0, I1.1...' | German: 'S1 254 Row 26 Switch Fault... Check Ixxx.x / Ixxx.x German' | French: 'S1 254 Row 26 Switch Fault... Check Ixxx.x / Ixxx.x French'
  255 = 'Spare' | German: 'S1 255 Row 26 Spare Message German' | French: 'S1 255 Row 26 Spare Message French'
  256 = 'Spare' | German: 'S1 256 Row 26 Spare Message German' | French: 'S1 256 Row 26 Spare Message French'
  257 = 'Spare' | German: 'S1 257 Row 26 Spare Message German' | French: 'S1 257 Row 26 Spare Message French'
  258 = 'Spare' | German: 'S1 258 Row 26 Spare Message German' | French: 'S1 258 Row 26 Spare Message French'
  259 = 'Spare' | German: 'S1 259 Row 26 Spare Message German' | French: 'S1 259 Row 26 Spare Message French'
  260 = 'Clamp Cylinder A1 Failed to Advance... Check Q1.0...' | German: 'S1 260 Row 27 Failed To Advance.. Check Qxxx.x German' | French: 'S1 260 Row 27 Failed To Advance.. Check Qxxx.x French'
  261 = 'Clamp Cylinder A1 Failed to Return... Check Q1.1...' | German: 'S1 261 Row 27 Failed To Return.. Check Qxxx.x German' | French: 'S1 261 Row 27 Failed To Return.. Check Qxxx.x French'
  262 = 'Clamp Cylinder A1 Lost Advanced... Check I1.0...' | German: 'S1 262 Row 27 Lost Advance Position... Check Ixxx.x German' | French: 'S1 262 Row 27 Lost Advance Position... Check Ixxx.x French'
  263 = 'Clamp Cylinder A1 Lost Returned... Check I1.1...' | German: 'S1 263 Row 27 Lost Return Position... Check Ixxx.x German' | French: 'S1 263 Row 27 Lost Return Position... Check Ixxx.x French'
  264 = 'Clamp Cylinder A1 Switch Fault... Check I1.0, I1.1...' | German: 'S1 264 Row 27 Switch Fault... Check Ixxx.x / Ixxx.x German' | French: 'S1 264 Row 27 Switch Fault... Check Ixxx.x / Ixxx.x French'
  265 = 'Spare' | German: 'S1 265 Row 27 Spare Message German' | French: 'S1 265 Row 27 Spare Message French'
  266 = 'Spare' | German: 'S1 266 Row 27 Spare Message German' | French: 'S1 266 Row 27 Spare Message French'
  267 = 'Spare' | German: 'S1 267 Row 27 Spare Message German' | French: 'S1 267 Row 27 Spare Message French'
  268 = 'Spare' | German: 'S1 268 Row 27 Spare Message German' | French: 'S1 268 Row 27 Spare Message French'
  269 = 'Spare' | German: 'S1 269 Row 27 Spare Message German' | French: 'S1 269 Row 27 Spare Message French'
  270 = 'Clamp Cylinder A1 Failed to Advance... Check Q1.0...' | German: 'S1 270 Row 28 Failed To Advance.. Check Qxxx.x German' | French: 'S1 270 Row 28 Failed To Advance.. Check Qxxx.x French'
  271 = 'Clamp Cylinder A1 Failed to Return... Check Q1.1...' | German: 'S1 271 Row 28 Failed To Return.. Check Qxxx.x German' | French: 'S1 271 Row 28 Failed To Return.. Check Qxxx.x French'
  272 = 'Clamp Cylinder A1 Lost Advanced... Check I1.0...' | German: 'S1 272 Row 28 Lost Advance Position... Check Ixxx.x German' | French: 'S1 272 Row 28 Lost Advance Position... Check Ixxx.x French'
  273 = 'Clamp Cylinder A1 Lost Returned... Check I1.1...' | German: 'S1 273 Row 28 Lost Return Position... Check Ixxx.x German' | French: 'S1 273 Row 28 Lost Return Position... Check Ixxx.x French'
  274 = 'Clamp Cylinder A1 Switch Fault... Check I1.0, I1.1...' | German: 'S1 274 Row 28 Switch Fault... Check Ixxx.x / Ixxx.x German' | French: 'S1 274 Row 28 Switch Fault... Check Ixxx.x / Ixxx.x French'
  275 = 'Spare' | German: 'S1 275 Row 28 Spare Message German' | French: 'S1 275 Row 28 Spare Message French'
  276 = 'Spare' | German: 'S1 276 Row 28 Spare Message German' | French: 'S1 276 Row 28 Spare Message French'
  277 = 'Spare' | German: 'S1 277 Row 28 Spare Message German' | French: 'S1 277 Row 28 Spare Message French'
  278 = 'Spare' | German: 'S1 278 Row 28 Spare Message German' | French: 'S1 278 Row 28 Spare Message French'
  279 = 'Spare' | German: 'S1 279 Row 28 Spare Message German' | French: 'S1 279 Row 28 Spare Message French'
  280 = 'Clamp Cylinder A1 Failed to Advance... Check Q1.0...' | German: 'S1 280 Row 29 Failed To Advance.. Check Qxxx.x German' | French: 'S1 280 Row 29 Failed To Advance.. Check Qxxx.x French'
  281 = 'Clamp Cylinder A1 Failed to Return... Check Q1.1...' | German: 'S1 281 Row 29 Failed To Return.. Check Qxxx.x German' | French: 'S1 281 Row 29 Failed To Return.. Check Qxxx.x French'
  282 = 'Clamp Cylinder A1 Lost Advanced... Check I1.0...' | German: 'S1 282 Row 29 Lost Advance Position... Check Ixxx.x German' | French: 'S1 282 Row 29 Lost Advance Position... Check Ixxx.x French'
  283 = 'Clamp Cylinder A1 Lost Returned... Check I1.1...' | German: 'S1 283 Row 29 Lost Return Position... Check Ixxx.x German' | French: 'S1 283 Row 29 Lost Return Position... Check Ixxx.x French'
  284 = 'Clamp Cylinder A1 Switch Fault... Check I1.0, I1.1...' | German: 'S1 284 Row 29 Switch Fault... Check Ixxx.x / Ixxx.x German' | French: 'S1 284 Row 29 Switch Fault... Check Ixxx.x / Ixxx.x French'
  285 = 'Spare' | German: 'S1 285 Row 29 Spare Message German' | French: 'S1 285 Row 29 Spare Message French'
  286 = 'Spare' | German: 'S1 286 Row 29 Spare Message German' | French: 'S1 286 Row 29 Spare Message French'
  287 = 'Spare' | German: 'S1 287 Row 29 Spare Message German' | French: 'S1 287 Row 29 Spare Message French'
  288 = 'Spare' | German: 'S1 288 Row 29 Spare Message German' | French: 'S1 288 Row 29 Spare Message French'
  289 = 'Spare' | German: 'S1 289 Row 29 Spare Message German' | French: 'S1 289 Row 29 Spare Message French'
  290 = 'Clamp Cylinder A1 Failed to Advance... Check Q1.0...' | German: 'S1 290 Row 30 Failed To Advance.. Check Qxxx.x German' | French: 'S1 290 Row 30 Failed To Advance.. Check Qxxx.x French'
  291 = 'Clamp Cylinder A1 Failed to Return... Check Q1.1...' | German: 'S1 291 Row 30 Failed To Return.. Check Qxxx.x German' | French: 'S1 291 Row 30 Failed To Return.. Check Qxxx.x French'
  292 = 'Clamp Cylinder A1 Lost Advanced... Check I1.0...' | German: 'S1 292 Row 30 Lost Advance Position... Check Ixxx.x German' | French: 'S1 292 Row 30 Lost Advance Position... Check Ixxx.x French'
  293 = 'Clamp Cylinder A1 Lost Returned... Check I1.1...' | German: 'S1 293 Row 30 Lost Return Position... Check Ixxx.x German' | French: 'S1 293 Row 30 Lost Return Position... Check Ixxx.x French'
  294 = 'Clamp Cylinder A1 Switch Fault... Check I1.0, I1.1...' | German: 'S1 294 Row 30 Switch Fault... Check Ixxx.x / Ixxx.x German' | French: 'S1 294 Row 30 Switch Fault... Check Ixxx.x / Ixxx.x French'
  295 = 'Spare' | German: 'S1 295 Row 30 Spare Message German' | French: 'S1 295 Row 30 Spare Message French'
  296 = 'Spare' | German: 'S1 296 Row 30 Spare Message German' | French: 'S1 296 Row 30 Spare Message French'
  297 = 'Spare' | German: 'S1 297 Row 30 Spare Message German' | French: 'S1 297 Row 30 Spare Message French'
  298 = 'Spare' | German: 'S1 298 Row 30 Spare Message German' | French: 'S1 298 Row 30 Spare Message French'
  299 = 'Spare' | German: 'S1 299 Row 30 Spare Message German' | French: 'S1 299 Row 30 Spare Message French'
  300 = 'Clamp Cylinder A1 Failed to Advance... Check Q1.0...' | German: 'S1 300 Row 31 Failed To Advance.. Check Qxxx.x German' | French: 'S1 300 Row 31 Failed To Advance.. Check Qxxx.x French'
  301 = 'Clamp Cylinder A1 Failed to Return... Check Q1.1...' | German: 'S1 301 Row 31 Failed To Return.. Check Qxxx.x German' | French: 'S1 301 Row 31 Failed To Return.. Check Qxxx.x French'
  302 = 'Clamp Cylinder A1 Lost Advanced... Check I1.0...' | German: 'S1 302 Row 31 Lost Advance Position... Check Ixxx.x German' | French: 'S1 302 Row 31 Lost Advance Position... Check Ixxx.x French'
  303 = 'Clamp Cylinder A1 Lost Returned... Check I1.1...' | German: 'S1 303 Row 31 Lost Return Position... Check Ixxx.x German' | French: 'S1 303 Row 31 Lost Return Position... Check Ixxx.x French'
  304 = 'Clamp Cylinder A1 Switch Fault... Check I1.0, I1.1...' | German: 'S1 304 Row 31 Switch Fault... Check Ixxx.x / Ixxx.x German' | French: 'S1 304 Row 31 Switch Fault... Check Ixxx.x / Ixxx.x French'
  305 = 'Spare' | German: 'S1 305 Row 31 Spare Message German' | French: 'S1 305 Row 31 Spare Message French'
  306 = 'Spare' | German: 'S1 306 Row 31 Spare Message German' | French: 'S1 306 Row 31 Spare Message French'
  307 = 'Spare' | German: 'S1 307 Row 31 Spare Message German' | French: 'S1 307 Row 31 Spare Message French'
  308 = 'Spare' | German: 'S1 308 Row 31 Spare Message German' | French: 'S1 308 Row 31 Spare Message French'
  309 = 'Spare' | German: 'S1 309 Row 31 Spare Message German' | French: 'S1 309 Row 31 Spare Message French'
  310 = 'Clamp Cylinder A1 Failed to Advance... Check Q1.0...' | German: 'S1 310 Row 32 Failed To Advance.. Check Qxxx.x German' | French: 'S1 310 Row 32 Failed To Advance.. Check Qxxx.x French'
  311 = 'Clamp Cylinder A1 Failed to Return... Check Q1.1...' | German: 'S1 311 Row 32 Failed To Return.. Check Qxxx.x German' | French: 'S1 311 Row 32 Failed To Return.. Check Qxxx.x French'
  312 = 'Clamp Cylinder A1 Lost Advanced... Check I1.0...' | German: 'S1 312 Row 32 Lost Advance Position... Check Ixxx.x German' | French: 'S1 312 Row 32 Lost Advance Position... Check Ixxx.x French'
  313 = 'Clamp Cylinder A1 Lost Returned... Check I1.1...' | German: 'S1 313 Row 32 Lost Return Position... Check Ixxx.x German' | French: 'S1 313 Row 32 Lost Return Position... Check Ixxx.x French'
  314 = 'Clamp Cylinder A1 Switch Fault... Check I1.0, I1.1...' | German: 'S1 314 Row 32 Switch Fault... Check Ixxx.x / Ixxx.x German' | French: 'S1 314 Row 32 Switch Fault... Check Ixxx.x / Ixxx.x French'
  315 = 'Spare' | German: 'S1 315 Row 32 Spare Message German' | French: 'S1 315 Row 32 Spare Message French'
  316 = 'Spare' | German: 'S1 316 Row 32 Spare Message German' | French: 'S1 316 Row 32 Spare Message French'
  317 = 'Spare' | German: 'S1 317 Row 32 Spare Message German' | French: 'S1 317 Row 32 Spare Message French'
  318 = 'Spare' | German: 'S1 318 Row 32 Spare Message German' | French: 'S1 318 Row 32 Spare Message French'
  319 = 'Spare' | German: 'S1 319 Row 32 Spare Message German' | French: 'S1 319 Row 32 Spare Message French'
  320 = 'Clamp Cylinder A1 Failed to Advance... Check Q1.0...' | German: 'S1 320 Row 33 Failed To Advance.. Check Qxxx.x German' | French: 'S1 320 Row 33 Failed To Advance.. Check Qxxx.x French'
  321 = 'Clamp Cylinder A1 Failed to Return... Check Q1.1...' | German: 'S1 321 Row 33 Failed To Return.. Check Qxxx.x German' | French: 'S1 321 Row 33 Failed To Return.. Check Qxxx.x French'
  322 = 'Clamp Cylinder A1 Lost Advanced... Check I1.0...' | German: 'S1 322 Row 33 Lost Advance Position... Check Ixxx.x German' | French: 'S1 322 Row 33 Lost Advance Position... Check Ixxx.x French'
  323 = 'Clamp Cylinder A1 Lost Returned... Check I1.1...' | German: 'S1 323 Row 33 Lost Return Position... Check Ixxx.x German' | French: 'S1 323 Row 33 Lost Return Position... Check Ixxx.x French'
  324 = 'Clamp Cylinder A1 Switch Fault... Check I1.0, I1.1...' | German: 'S1 324 Row 33 Switch Fault... Check Ixxx.x / Ixxx.x German' | French: 'S1 324 Row 33 Switch Fault... Check Ixxx.x / Ixxx.x French'
  325 = 'Spare' | German: 'S1 325 Row 33 Spare Message German' | French: 'S1 325 Row 33 Spare Message French'
  326 = 'Spare' | German: 'S1 326 Row 33 Spare Message German' | French: 'S1 326 Row 33 Spare Message French'
  327 = 'Spare' | German: 'S1 327 Row 33 Spare Message German' | French: 'S1 327 Row 33 Spare Message French'
  328 = 'Spare' | German: 'S1 328 Row 33 Spare Message German' | French: 'S1 328 Row 33 Spare Message French'
  329 = 'Spare' | German: 'S1 329 Row 33 Spare Message German' | French: 'S1 329 Row 33 Spare Message French'
  330 = 'Clamp Cylinder A1 Failed to Advance... Check Q1.0...' | German: 'S1 330 Row 34 Failed To Advance.. Check Qxxx.x German' | French: 'S1 330 Row 34 Failed To Advance.. Check Qxxx.x French'
  331 = 'Clamp Cylinder A1 Failed to Return... Check Q1.1...' | German: 'S1 331 Row 34 Failed To Return.. Check Qxxx.x German' | French: 'S1 331 Row 34 Failed To Return.. Check Qxxx.x French'
  332 = 'Clamp Cylinder A1 Lost Advanced... Check I1.0...' | German: 'S1 332 Row 34 Lost Advance Position... Check Ixxx.x German' | French: 'S1 332 Row 34 Lost Advance Position... Check Ixxx.x French'
  333 = 'Clamp Cylinder A1 Lost Returned... Check I1.1...' | German: 'S1 333 Row 34 Lost Return Position... Check Ixxx.x German' | French: 'S1 333 Row 34 Lost Return Position... Check Ixxx.x French'
  334 = 'Clamp Cylinder A1 Switch Fault... Check I1.0, I1.1...' | German: 'S1 334 Row 34 Switch Fault... Check Ixxx.x / Ixxx.x German' | French: 'S1 334 Row 34 Switch Fault... Check Ixxx.x / Ixxx.x French'
  335 = 'Spare' | German: 'S1 335 Row 34 Spare Message German' | French: 'S1 335 Row 34 Spare Message French'
  336 = 'Spare' | German: 'S1 336 Row 34 Spare Message German' | French: 'S1 336 Row 34 Spare Message French'
  337 = 'Spare' | German: 'S1 337 Row 34 Spare Message German' | French: 'S1 337 Row 34 Spare Message French'
  338 = 'Spare' | German: 'S1 338 Row 34 Spare Message German' | French: 'S1 338 Row 34 Spare Message French'
  339 = 'Spare' | German: 'S1 339 Row 34 Spare Message German' | French: 'S1 339 Row 34 Spare Message French'
  340 = 'Clamp Cylinder A1 Failed to Advance... Check Q1.0...' | German: 'S1 340 Row 35 Failed To Advance.. Check Qxxx.x German' | French: 'S1 340 Row 35 Failed To Advance.. Check Qxxx.x French'
  341 = 'Clamp Cylinder A1 Failed to Return... Check Q1.1...' | German: 'S1 341 Row 35 Failed To Return.. Check Qxxx.x German' | French: 'S1 341 Row 35 Failed To Return.. Check Qxxx.x French'
  342 = 'Clamp Cylinder A1 Lost Advanced... Check I1.0...' | German: 'S1 342 Row 35 Lost Advance Position... Check Ixxx.x German' | French: 'S1 342 Row 35 Lost Advance Position... Check Ixxx.x French'
  343 = 'Clamp Cylinder A1 Lost Returned... Check I1.1...' | German: 'S1 343 Row 35 Lost Return Position... Check Ixxx.x German' | French: 'S1 343 Row 35 Lost Return Position... Check Ixxx.x French'
  344 = 'Clamp Cylinder A1 Switch Fault... Check I1.0, I1.1...' | German: 'S1 344 Row 35 Switch Fault... Check Ixxx.x / Ixxx.x German' | French: 'S1 344 Row 35 Switch Fault... Check Ixxx.x / Ixxx.x French'
  345 = 'Spare' | German: 'S1 345 Row 35 Spare Message German' | French: 'S1 345 Row 35 Spare Message French'
  346 = 'Spare' | German: 'S1 346 Row 35 Spare Message German' | French: 'S1 346 Row 35 Spare Message French'
  347 = 'Spare' | German: 'S1 347 Row 35 Spare Message German' | French: 'S1 347 Row 35 Spare Message French'
  348 = 'Spare' | German: 'S1 348 Row 35 Spare Message German' | French: 'S1 348 Row 35 Spare Message French'
  349 = 'Spare' | German: 'S1 349 Row 35 Spare Message German' | French: 'S1 349 Row 35 Spare Message French'
  350 = 'Clamp Cylinder A1 Failed to Advance... Check Q1.0...' | German: 'S1 350 Row 36 Failed To Advance.. Check Qxxx.x German' | French: 'S1 350 Row 36 Failed To Advance.. Check Qxxx.x French'
  351 = 'Clamp Cylinder A1 Failed to Return... Check Q1.1...' | German: 'S1 351 Row 36 Failed To Return.. Check Qxxx.x German' | French: 'S1 351 Row 36 Failed To Return.. Check Qxxx.x French'
  352 = 'Clamp Cylinder A1 Lost Advanced... Check I1.0...' | German: 'S1 352 Row 36 Lost Advance Position... Check Ixxx.x German' | French: 'S1 352 Row 36 Lost Advance Position... Check Ixxx.x French'
  353 = 'Clamp Cylinder A1 Lost Returned... Check I1.1...' | German: 'S1 353 Row 36 Lost Return Position... Check Ixxx.x German' | French: 'S1 353 Row 36 Lost Return Position... Check Ixxx.x French'
  354 = 'Clamp Cylinder A1 Switch Fault... Check I1.0, I1.1...' | German: 'S1 354 Row 36 Switch Fault... Check Ixxx.x / Ixxx.x German' | French: 'S1 354 Row 36 Switch Fault... Check Ixxx.x / Ixxx.x French'
  355 = 'Spare' | German: 'S1 355 Row 36 Spare Message German' | French: 'S1 355 Row 36 Spare Message French'
  356 = 'Spare' | German: 'S1 356 Row 36 Spare Message German' | French: 'S1 356 Row 36 Spare Message French'
  357 = 'Spare' | German: 'S1 357 Row 36 Spare Message German' | French: 'S1 357 Row 36 Spare Message French'
  358 = 'Spare' | German: 'S1 358 Row 36 Spare Message German' | French: 'S1 358 Row 36 Spare Message French'
  359 = 'Spare' | German: 'S1 359 Row 36 Spare Message German' | French: 'S1 359 Row 36 Spare Message French'
  360 = 'Clamp Cylinder A1 Failed to Advance... Check Q1.0...' | German: 'S1 360 Row 37 Failed To Advance.. Check Qxxx.x German' | French: 'S1 360 Row 37 Failed To Advance.. Check Qxxx.x French'
  361 = 'Clamp Cylinder A1 Failed to Return... Check Q1.1...' | German: 'S1 361 Row 37 Failed To Return.. Check Qxxx.x German' | French: 'S1 361 Row 37 Failed To Return.. Check Qxxx.x French'
  362 = 'Clamp Cylinder A1 Lost Advanced... Check I1.0...' | German: 'S1 362 Row 37 Lost Advance Position... Check Ixxx.x German' | French: 'S1 362 Row 37 Lost Advance Position... Check Ixxx.x French'
  363 = 'Clamp Cylinder A1 Lost Returned... Check I1.1...' | German: 'S1 363 Row 37 Lost Return Position... Check Ixxx.x German' | French: 'S1 363 Row 37 Lost Return Position... Check Ixxx.x French'
  364 = 'Clamp Cylinder A1 Switch Fault... Check I1.0, I1.1...' | German: 'S1 364 Row 37 Switch Fault... Check Ixxx.x / Ixxx.x German' | French: 'S1 364 Row 37 Switch Fault... Check Ixxx.x / Ixxx.x French'
  365 = 'Spare' | German: 'S1 365 Row 37 Spare Message German' | French: 'S1 365 Row 37 Spare Message French'
  366 = 'Spare' | German: 'S1 366 Row 37 Spare Message German' | French: 'S1 366 Row 37 Spare Message French'
  367 = 'Spare' | German: 'S1 367 Row 37 Spare Message German' | French: 'S1 367 Row 37 Spare Message French'
  368 = 'Spare' | German: 'S1 368 Row 37 Spare Message German' | French: 'S1 368 Row 37 Spare Message French'
  369 = 'Spare' | German: 'S1 369 Row 37 Spare Message German' | French: 'S1 369 Row 37 Spare Message French'
  370 = 'Clamp Cylinder A1 Failed to Advance... Check Q1.0...' | German: 'S1 370 Row 38 Failed To Advance.. Check Qxxx.x German' | French: 'S1 370 Row 38 Failed To Advance.. Check Qxxx.x French'
  371 = 'Clamp Cylinder A1 Failed to Return... Check Q1.1...' | German: 'S1 371 Row 38 Failed To Return.. Check Qxxx.x German' | French: 'S1 371 Row 38 Failed To Return.. Check Qxxx.x French'
  372 = 'Clamp Cylinder A1 Lost Advanced... Check I1.0...' | German: 'S1 372 Row 38 Lost Advance Position... Check Ixxx.x German' | French: 'S1 372 Row 38 Lost Advance Position... Check Ixxx.x French'
  373 = 'Clamp Cylinder A1 Lost Returned... Check I1.1...' | German: 'S1 373 Row 38 Lost Return Position... Check Ixxx.x German' | French: 'S1 373 Row 38 Lost Return Position... Check Ixxx.x French'
  374 = 'Clamp Cylinder A1 Switch Fault... Check I1.0, I1.1...' | German: 'S1 374 Row 38 Switch Fault... Check Ixxx.x / Ixxx.x German' | French: 'S1 374 Row 38 Switch Fault... Check Ixxx.x / Ixxx.x French'
  375 = 'Spare' | German: 'S1 375 Row 38 Spare Message German' | French: 'S1 375 Row 38 Spare Message French'
  376 = 'Spare' | German: 'S1 376 Row 38 Spare Message German' | French: 'S1 376 Row 38 Spare Message French'
  377 = 'Spare' | German: 'S1 377 Row 38 Spare Message German' | French: 'S1 377 Row 38 Spare Message French'
  378 = 'Spare' | German: 'S1 378 Row 38 Spare Message German' | French: 'S1 378 Row 38 Spare Message French'
  379 = 'Spare' | German: 'S1 379 Row 38 Spare Message German' | French: 'S1 379 Row 38 Spare Message French'
  380 = 'Clamp Cylinder A1 Failed to Advance... Check Q1.0...' | German: 'S1 380 Row 39 Failed To Advance.. Check Qxxx.x German' | French: 'S1 380 Row 39 Failed To Advance.. Check Qxxx.x French'
  381 = 'Clamp Cylinder A1 Failed to Return... Check Q1.1...' | German: 'S1 381 Row 39 Failed To Return.. Check Qxxx.x German' | French: 'S1 381 Row 39 Failed To Return.. Check Qxxx.x French'
  382 = 'Clamp Cylinder A1 Lost Advanced... Check I1.0...' | German: 'S1 382 Row 39 Lost Advance Position... Check Ixxx.x German' | French: 'S1 382 Row 39 Lost Advance Position... Check Ixxx.x French'
  383 = 'Clamp Cylinder A1 Lost Returned... Check I1.1...' | German: 'S1 383 Row 39 Lost Return Position... Check Ixxx.x German' | French: 'S1 383 Row 39 Lost Return Position... Check Ixxx.x French'
  384 = 'Clamp Cylinder A1 Switch Fault... Check I1.0, I1.1...' | German: 'S1 384 Row 39 Switch Fault... Check Ixxx.x / Ixxx.x German' | French: 'S1 384 Row 39 Switch Fault... Check Ixxx.x / Ixxx.x French'
  385 = 'Spare' | German: 'S1 385 Row 39 Spare Message German' | French: 'S1 385 Row 39 Spare Message French'
  386 = 'Spare' | German: 'S1 386 Row 39 Spare Message German' | French: 'S1 386 Row 39 Spare Message French'
  387 = 'Spare' | German: 'S1 387 Row 39 Spare Message German' | French: 'S1 387 Row 39 Spare Message French'
  388 = 'Spare' | German: 'S1 388 Row 39 Spare Message German' | French: 'S1 388 Row 39 Spare Message French'
  389 = 'Spare' | German: 'S1 389 Row 39 Spare Message German' | French: 'S1 389 Row 39 Spare Message French'
  390 = 'Clamp Cylinder A1 Failed to Advance... Check Q1.0...' | German: 'S1 390 Row 40 Failed To Advance.. Check Qxxx.x German' | French: 'S1 390 Row 40 Failed To Advance.. Check Qxxx.x French'
  391 = 'Clamp Cylinder A1 Failed to Return... Check Q1.1...' | German: 'S1 391 Row 40 Failed To Return.. Check Qxxx.x German' | French: 'S1 391 Row 40 Failed To Return.. Check Qxxx.x French'
  392 = 'Clamp Cylinder A1 Lost Advanced... Check I1.0...' | German: 'S1 392 Row 40 Lost Advance Position... Check Ixxx.x German' | French: 'S1 392 Row 40 Lost Advance Position... Check Ixxx.x French'
  393 = 'Clamp Cylinder A1 Lost Returned... Check I1.1...' | German: 'S1 393 Row 40 Lost Return Position... Check Ixxx.x German' | French: 'S1 393 Row 40 Lost Return Position... Check Ixxx.x French'
  394 = 'Clamp Cylinder A1 Switch Fault... Check I1.0, I1.1...' | German: 'S1 394 Row 40 Switch Fault... Check Ixxx.x / Ixxx.x German' | French: 'S1 394 Row 40 Switch Fault... Check Ixxx.x / Ixxx.x French'
  395 = 'Spare' | German: 'S1 395 Row 40 Spare Message German' | French: 'S1 395 Row 40 Spare Message French'
  396 = 'Spare' | German: 'S1 396 Row 40 Spare Message German' | French: 'S1 396 Row 40 Spare Message French'
  397 = 'Spare' | German: 'S1 397 Row 40 Spare Message German' | French: 'S1 397 Row 40 Spare Message French'
  398 = 'Spare' | German: 'S1 398 Row 40 Spare Message German' | French: 'S1 398 Row 40 Spare Message French'
  399 = 'Spare' | German: 'S1 399 Row 40 Spare Message German' | French: 'S1 399 Row 40 Spare Message French'
  400 = 'Clamp Cylinder A1 Failed to Advance... Check Q1.0...' | German: 'S1 400 Row 41 Failed To Advance.. Check Qxxx.x German' | French: 'S1 400 Row 41 Failed To Advance.. Check Qxxx.x French'
  401 = 'Clamp Cylinder A1 Failed to Return... Check Q1.1...' | German: 'S1 401 Row 41 Failed To Return.. Check Qxxx.x German' | French: 'S1 401 Row 41 Failed To Return.. Check Qxxx.x French'
  402 = 'Clamp Cylinder A1 Lost Advanced... Check I1.0...' | German: 'S1 402 Row 41 Lost Advance Position... Check Ixxx.x German' | French: 'S1 402 Row 41 Lost Advance Position... Check Ixxx.x French'
  403 = 'Clamp Cylinder A1 Lost Returned... Check I1.1...' | German: 'S1 403 Row 41 Lost Return Position... Check Ixxx.x German' | French: 'S1 403 Row 41 Lost Return Position... Check Ixxx.x French'
  404 = 'Clamp Cylinder A1 Switch Fault... Check I1.0, I1.1...' | German: 'S1 404 Row 41 Switch Fault... Check Ixxx.x / Ixxx.x German' | French: 'S1 404 Row 41 Switch Fault... Check Ixxx.x / Ixxx.x French'
  405 = 'Spare' | German: 'S1 405 Row 41 Spare Message German' | French: 'S1 405 Row 41 Spare Message French'
  406 = 'Spare' | German: 'S1 406 Row 41 Spare Message German' | French: 'S1 406 Row 41 Spare Message French'
  407 = 'Spare' | German: 'S1 407 Row 41 Spare Message German' | French: 'S1 407 Row 41 Spare Message French'
  408 = 'Spare' | German: 'S1 408 Row 41 Spare Message German' | French: 'S1 408 Row 41 Spare Message French'
  409 = 'Spare' | German: 'S1 409 Row 41 Spare Message German' | French: 'S1 409 Row 41 Spare Message French'
  410 = 'Clamp Cylinder A1 Failed to Advance... Check Q1.0...' | German: 'S1 410 Row 42 Failed To Advance.. Check Qxxx.x German' | French: 'S1 410 Row 42 Failed To Advance.. Check Qxxx.x French'
  411 = 'Clamp Cylinder A1 Failed to Return... Check Q1.1...' | German: 'S1 411 Row 42 Failed To Return.. Check Qxxx.x German' | French: 'S1 411 Row 42 Failed To Return.. Check Qxxx.x French'
  412 = 'Clamp Cylinder A1 Lost Advanced... Check I1.0...' | German: 'S1 412 Row 42 Lost Advance Position... Check Ixxx.x German' | French: 'S1 412 Row 42 Lost Advance Position... Check Ixxx.x French'
  413 = 'Clamp Cylinder A1 Lost Returned... Check I1.1...' | German: 'S1 413 Row 42 Lost Return Position... Check Ixxx.x German' | French: 'S1 413 Row 42 Lost Return Position... Check Ixxx.x French'
  414 = 'Clamp Cylinder A1 Switch Fault... Check I1.0, I1.1...' | German: 'S1 414 Row 42 Switch Fault... Check Ixxx.x / Ixxx.x German' | French: 'S1 414 Row 42 Switch Fault... Check Ixxx.x / Ixxx.x French'
  415 = 'Spare' | German: 'S1 415 Row 42 Spare Message German' | French: 'S1 415 Row 42 Spare Message French'
  416 = 'Spare' | German: 'S1 416 Row 42 Spare Message German' | French: 'S1 416 Row 42 Spare Message French'
  417 = 'Spare' | German: 'S1 417 Row 42 Spare Message German' | French: 'S1 417 Row 42 Spare Message French'
  418 = 'Spare' | German: 'S1 418 Row 42 Spare Message German' | French: 'S1 418 Row 42 Spare Message French'
  419 = 'Spare' | German: 'S1 419 Row 42 Spare Message German' | French: 'S1 419 Row 42 Spare Message French'
  420 = 'Clamp Cylinder A1 Failed to Advance... Check Q1.0...' | German: 'S1 420 Row 43 Failed To Advance.. Check Qxxx.x German' | French: 'S1 420 Row 43 Failed To Advance.. Check Qxxx.x French'
  421 = 'Clamp Cylinder A1 Failed to Return... Check Q1.1...' | German: 'S1 421 Row 43 Failed To Return.. Check Qxxx.x German' | French: 'S1 421 Row 43 Failed To Return.. Check Qxxx.x French'
  422 = 'Clamp Cylinder A1 Lost Advanced... Check I1.0...' | German: 'S1 422 Row 43 Lost Advance Position... Check Ixxx.x German' | French: 'S1 422 Row 43 Lost Advance Position... Check Ixxx.x French'
  423 = 'Clamp Cylinder A1 Lost Returned... Check I1.1...' | German: 'S1 423 Row 43 Lost Return Position... Check Ixxx.x German' | French: 'S1 423 Row 43 Lost Return Position... Check Ixxx.x French'
  424 = 'Clamp Cylinder A1 Switch Fault... Check I1.0, I1.1...' | German: 'S1 424 Row 43 Switch Fault... Check Ixxx.x / Ixxx.x German' | French: 'S1 424 Row 43 Switch Fault... Check Ixxx.x / Ixxx.x French'
  425 = 'Spare' | German: 'S1 425 Row 43 Spare Message German' | French: 'S1 425 Row 43 Spare Message French'
  426 = 'Spare' | German: 'S1 426 Row 43 Spare Message German' | French: 'S1 426 Row 43 Spare Message French'
  427 = 'Spare' | German: 'S1 427 Row 43 Spare Message German' | French: 'S1 427 Row 43 Spare Message French'
  428 = 'Spare' | German: 'S1 428 Row 43 Spare Message German' | French: 'S1 428 Row 43 Spare Message French'
  429 = 'Spare' | German: 'S1 429 Row 43 Spare Message German' | French: 'S1 429 Row 43 Spare Message French'
  430 = 'Clamp Cylinder A1 Failed to Advance... Check Q1.0...' | German: 'S1 430 Row 44 Failed To Advance.. Check Qxxx.x German' | French: 'S1 430 Row 44 Failed To Advance.. Check Qxxx.x French'
  431 = 'Clamp Cylinder A1 Failed to Return... Check Q1.1...' | German: 'S1 431 Row 44 Failed To Return.. Check Qxxx.x German' | French: 'S1 431 Row 44 Failed To Return.. Check Qxxx.x French'
  432 = 'Clamp Cylinder A1 Lost Advanced... Check I1.0...' | German: 'S1 432 Row 44 Lost Advance Position... Check Ixxx.x German' | French: 'S1 432 Row 44 Lost Advance Position... Check Ixxx.x French'
  433 = 'Clamp Cylinder A1 Lost Returned... Check I1.1...' | German: 'S1 433 Row 44 Lost Return Position... Check Ixxx.x German' | French: 'S1 433 Row 44 Lost Return Position... Check Ixxx.x French'
  434 = 'Clamp Cylinder A1 Switch Fault... Check I1.0, I1.1...' | German: 'S1 434 Row 44 Switch Fault... Check Ixxx.x / Ixxx.x German' | French: 'S1 434 Row 44 Switch Fault... Check Ixxx.x / Ixxx.x French'
  435 = 'Spare' | German: 'S1 435 Row 44 Spare Message German' | French: 'S1 435 Row 44 Spare Message French'
  436 = 'Spare' | German: 'S1 436 Row 44 Spare Message German' | French: 'S1 436 Row 44 Spare Message French'
  437 = 'Spare' | German: 'S1 437 Row 44 Spare Message German' | French: 'S1 437 Row 44 Spare Message French'
  438 = 'Spare' | German: 'S1 438 Row 44 Spare Message German' | French: 'S1 438 Row 44 Spare Message French'
  439 = 'Spare' | German: 'S1 439 Row 44 Spare Message German' | French: 'S1 439 Row 44 Spare Message French'
  440 = 'Clamp Cylinder A1 Failed to Advance... Check Q1.0...' | German: 'S1 440 Row 45 Failed To Advance.. Check Qxxx.x German' | French: 'S1 440 Row 45 Failed To Advance.. Check Qxxx.x French'
  441 = 'Clamp Cylinder A1 Failed to Return... Check Q1.1...' | German: 'S1 441 Row 45 Failed To Return.. Check Qxxx.x German' | French: 'S1 441 Row 45 Failed To Return.. Check Qxxx.x French'
  442 = 'Clamp Cylinder A1 Lost Advanced... Check I1.0...' | German: 'S1 442 Row 45 Lost Advance Position... Check Ixxx.x German' | French: 'S1 442 Row 45 Lost Advance Position... Check Ixxx.x French'
  443 = 'Clamp Cylinder A1 Lost Returned... Check I1.1...' | German: 'S1 443 Row 45 Lost Return Position... Check Ixxx.x German' | French: 'S1 443 Row 45 Lost Return Position... Check Ixxx.x French'
  444 = 'Clamp Cylinder A1 Switch Fault... Check I1.0, I1.1...' | German: 'S1 444 Row 45 Switch Fault... Check Ixxx.x / Ixxx.x German' | French: 'S1 444 Row 45 Switch Fault... Check Ixxx.x / Ixxx.x French'
  445 = 'Spare' | German: 'S1 445 Row 45 Spare Message German' | French: 'S1 445 Row 45 Spare Message French'
  446 = 'Spare' | German: 'S1 446 Row 45 Spare Message German' | French: 'S1 446 Row 45 Spare Message French'
  447 = 'Spare' | German: 'S1 447 Row 45 Spare Message German' | French: 'S1 447 Row 45 Spare Message French'
  448 = 'Spare' | German: 'S1 448 Row 45 Spare Message German' | French: 'S1 448 Row 45 Spare Message French'
  449 = 'Spare' | German: 'S1 449 Row 45 Spare Message German' | French: 'S1 449 Row 45 Spare Message French'
  450 = 'Clamp Cylinder A1 Failed to Advance... Check Q1.0...' | German: 'S1 450 Row 46 Failed To Advance.. Check Qxxx.x German' | French: 'S1 450 Row 46 Failed To Advance.. Check Qxxx.x French'
  451 = 'Clamp Cylinder A1 Failed to Return... Check Q1.1...' | German: 'S1 451 Row 46 Failed To Return.. Check Qxxx.x German' | French: 'S1 451 Row 46 Failed To Return.. Check Qxxx.x French'
  452 = 'Clamp Cylinder A1 Lost Advanced... Check I1.0...' | German: 'S1 452 Row 46 Lost Advance Position... Check Ixxx.x German' | French: 'S1 452 Row 46 Lost Advance Position... Check Ixxx.x French'
  453 = 'Clamp Cylinder A1 Lost Returned... Check I1.1...' | German: 'S1 453 Row 46 Lost Return Position... Check Ixxx.x German' | French: 'S1 453 Row 46 Lost Return Position... Check Ixxx.x French'
  454 = 'Clamp Cylinder A1 Switch Fault... Check I1.0, I1.1...' | German: 'S1 454 Row 46 Switch Fault... Check Ixxx.x / Ixxx.x German' | French: 'S1 454 Row 46 Switch Fault... Check Ixxx.x / Ixxx.x French'
  455 = 'Spare' | German: 'S1 455 Row 46 Spare Message German' | French: 'S1 455 Row 46 Spare Message French'
  456 = 'Spare' | German: 'S1 456 Row 46 Spare Message German' | French: 'S1 456 Row 46 Spare Message French'
  457 = 'Spare' | German: 'S1 457 Row 46 Spare Message German' | French: 'S1 457 Row 46 Spare Message French'
  458 = 'Spare' | German: 'S1 458 Row 46 Spare Message German' | French: 'S1 458 Row 46 Spare Message French'
  459 = 'Spare' | German: 'S1 459 Row 46 Spare Message German' | French: 'S1 459 Row 46 Spare Message French'
  460 = 'Clamp Cylinder A1 Failed to Advance... Check Q1.0...' | German: 'S1 460 Row 47 Failed To Advance.. Check Qxxx.x German' | French: 'S1 460 Row 47 Failed To Advance.. Check Qxxx.x French'
  461 = 'Clamp Cylinder A1 Failed to Return... Check Q1.1...' | German: 'S1 461 Row 47 Failed To Return.. Check Qxxx.x German' | French: 'S1 461 Row 47 Failed To Return.. Check Qxxx.x French'
  462 = 'Clamp Cylinder A1 Lost Advanced... Check I1.0...' | German: 'S1 462 Row 47 Lost Advance Position... Check Ixxx.x German' | French: 'S1 462 Row 47 Lost Advance Position... Check Ixxx.x French'
  463 = 'Clamp Cylinder A1 Lost Returned... Check I1.1...' | German: 'S1 463 Row 47 Lost Return Position... Check Ixxx.x German' | French: 'S1 463 Row 47 Lost Return Position... Check Ixxx.x French'
  464 = 'Clamp Cylinder A1 Switch Fault... Check I1.0, I1.1...' | German: 'S1 464 Row 47 Switch Fault... Check Ixxx.x / Ixxx.x German' | French: 'S1 464 Row 47 Switch Fault... Check Ixxx.x / Ixxx.x French'
  465 = 'Spare' | German: 'S1 465 Row 47 Spare Message German' | French: 'S1 465 Row 47 Spare Message French'
  466 = 'Spare' | German: 'S1 466 Row 47 Spare Message German' | French: 'S1 466 Row 47 Spare Message French'
  467 = 'Spare' | German: 'S1 467 Row 47 Spare Message German' | French: 'S1 467 Row 47 Spare Message French'
  468 = 'Spare' | German: 'S1 468 Row 47 Spare Message German' | French: 'S1 468 Row 47 Spare Message French'
  469 = 'Spare' | German: 'S1 469 Row 47 Spare Message German' | French: 'S1 469 Row 47 Spare Message French'
  470 = 'Clamp Cylinder A1 Failed to Advance... Check Q1.0...' | German: 'S1 470 Row 48 Failed To Advance.. Check Qxxx.x German' | French: 'S1 470 Row 48 Failed To Advance.. Check Qxxx.x French'
  471 = 'Clamp Cylinder A1 Failed to Return... Check Q1.1...' | German: 'S1 471 Row 48 Failed To Return.. Check Qxxx.x German' | French: 'S1 471 Row 48 Failed To Return.. Check Qxxx.x French'
  472 = 'Clamp Cylinder A1 Lost Advanced... Check I1.0...' | German: 'S1 472 Row 48 Lost Advance Position... Check Ixxx.x German' | French: 'S1 472 Row 48 Lost Advance Position... Check Ixxx.x French'
  473 = 'Clamp Cylinder A1 Lost Returned... Check I1.1...' | German: 'S1 473 Row 48 Lost Return Position... Check Ixxx.x German' | French: 'S1 473 Row 48 Lost Return Position... Check Ixxx.x French'
  474 = 'Clamp Cylinder A1 Switch Fault... Check I1.0, I1.1...' | German: 'S1 474 Row 48 Switch Fault... Check Ixxx.x / Ixxx.x German' | French: 'S1 474 Row 48 Switch Fault... Check Ixxx.x / Ixxx.x French'
  475 = 'Spare' | German: 'S1 475 Row 48 Spare Message German' | French: 'S1 475 Row 48 Spare Message French'
  476 = 'Spare' | German: 'S1 476 Row 48 Spare Message German' | French: 'S1 476 Row 48 Spare Message French'
  477 = 'Spare' | German: 'S1 477 Row 48 Spare Message German' | French: 'S1 477 Row 48 Spare Message French'
  478 = 'Spare' | German: 'S1 478 Row 48 Spare Message German' | French: 'S1 478 Row 48 Spare Message French'
  479 = 'Spare' | German: 'S1 479 Row 48 Spare Message German' | French: 'S1 479 Row 48 Spare Message French'
  480 = 'Clamp Cylinder A1 Failed to Advance... Check Q1.0...' | German: 'S1 480 Row 49 Failed To Advance.. Check Qxxx.x German' | French: 'S1 480 Row 49 Failed To Advance.. Check Qxxx.x French'
  481 = 'Clamp Cylinder A1 Failed to Return... Check Q1.1...' | German: 'S1 481 Row 49 Failed To Return.. Check Qxxx.x German' | French: 'S1 481 Row 49 Failed To Return.. Check Qxxx.x French'
  482 = 'Clamp Cylinder A1 Lost Advanced... Check I1.0...' | German: 'S1 482 Row 49 Lost Advance Position... Check Ixxx.x German' | French: 'S1 482 Row 49 Lost Advance Position... Check Ixxx.x French'
  483 = 'Clamp Cylinder A1 Lost Returned... Check I1.1...' | German: 'S1 483 Row 49 Lost Return Position... Check Ixxx.x German' | French: 'S1 483 Row 49 Lost Return Position... Check Ixxx.x French'
  484 = 'Clamp Cylinder A1 Switch Fault... Check I1.0, I1.1...' | German: 'S1 484 Row 49 Switch Fault... Check Ixxx.x / Ixxx.x German' | French: 'S1 484 Row 49 Switch Fault... Check Ixxx.x / Ixxx.x French'
  485 = 'Spare' | German: 'S1 485 Row 49 Spare Message German' | French: 'S1 485 Row 49 Spare Message French'
  486 = 'Spare' | German: 'S1 486 Row 49 Spare Message German' | French: 'S1 486 Row 49 Spare Message French'
  487 = 'Spare' | German: 'S1 487 Row 49 Spare Message German' | French: 'S1 487 Row 49 Spare Message French'
  488 = 'Spare' | German: 'S1 488 Row 49 Spare Message German' | French: 'S1 488 Row 49 Spare Message French'
  489 = 'Spare' | German: 'S1 489 Row 49 Spare Message German' | French: 'S1 489 Row 49 Spare Message French'
  490 = 'Clamp Cylinder A1 Failed to Advance... Check Q1.0...' | German: 'S1 490 Row 50 Failed To Advance.. Check Qxxx.x German' | French: 'S1 490 Row 50 Failed To Advance.. Check Qxxx.x French'
  491 = 'Clamp Cylinder A1 Failed to Return... Check Q1.1...' | German: 'S1 491 Row 50 Failed To Return.. Check Qxxx.x German' | French: 'S1 491 Row 50 Failed To Return.. Check Qxxx.x French'
  492 = 'Clamp Cylinder A1 Lost Advanced... Check I1.0...' | German: 'S1 492 Row 50 Lost Advance Position... Check Ixxx.x German' | French: 'S1 492 Row 50 Lost Advance Position... Check Ixxx.x French'
  493 = 'Clamp Cylinder A1 Lost Returned... Check I1.1...' | German: 'S1 493 Row 50 Lost Return Position... Check Ixxx.x German' | French: 'S1 493 Row 50 Lost Return Position... Check Ixxx.x French'
  494 = 'Clamp Cylinder A1 Switch Fault... Check I1.0, I1.1...' | German: 'S1 494 Row 50 Switch Fault... Check Ixxx.x / Ixxx.x German' | French: 'S1 494 Row 50 Switch Fault... Check Ixxx.x / Ixxx.x French'
  495 = 'Spare' | German: 'S1 495 Row 50 Spare Message German' | French: 'S1 495 Row 50 Spare Message French'
  496 = 'Spare' | German: 'S1 496 Row 50 Spare Message German' | French: 'S1 496 Row 50 Spare Message French'
  497 = 'Spare' | German: 'S1 497 Row 50 Spare Message German' | French: 'S1 497 Row 50 Spare Message French'
  498 = 'Spare' | German: 'S1 498 Row 50 Spare Message German' | French: 'S1 498 Row 50 Spare Message French'
  499 = 'Spare' | German: 'S1 499 Row 50 Spare Message German' | French: 'S1 499 Row 50 Spare Message French'
  500 = 'Clamp Cylinder A1 Failed to Advance... Check Q1.0...' | German: 'S1 500 Row 51 Failed To Advance.. Check Qxxx.x German' | French: 'S1 500 Row 51 Failed To Advance.. Check Qxxx.x French'
  501 = 'Clamp Cylinder A1 Failed to Return... Check Q1.1...' | German: 'S1 501 Row 51 Failed To Return.. Check Qxxx.x German' | French: 'S1 501 Row 51 Failed To Return.. Check Qxxx.x French'
  502 = 'Clamp Cylinder A1 Lost Advanced... Check I1.0...' | German: 'S1 502 Row 51 Lost Advance Position... Check Ixxx.x German' | French: 'S1 502 Row 51 Lost Advance Position... Check Ixxx.x French'
  503 = 'Clamp Cylinder A1 Lost Returned... Check I1.1...' | German: 'S1 503 Row 51 Lost Return Position... Check Ixxx.x German' | French: 'S1 503 Row 51 Lost Return Position... Check Ixxx.x French'
  504 = 'Clamp Cylinder A1 Switch Fault... Check I1.0, I1.1...' | German: 'S1 504 Row 51 Switch Fault... Check Ixxx.x / Ixxx.x German' | French: 'S1 504 Row 51 Switch Fault... Check Ixxx.x / Ixxx.x French'
  505 = 'Spare' | German: 'S1 505 Row 51 Spare Message German' | French: 'S1 505 Row 51 Spare Message French'
  506 = 'Spare' | German: 'S1 506 Row 51 Spare Message German' | French: 'S1 506 Row 51 Spare Message French'
  507 = 'Spare' | German: 'S1 507 Row 51 Spare Message German' | French: 'S1 507 Row 51 Spare Message French'
  508 = 'Spare' | German: 'S1 508 Row 51 Spare Message German' | French: 'S1 508 Row 51 Spare Message French'
  509 = 'Spare' | German: 'S1 509 Row 51 Spare Message German' | French: 'S1 509 Row 51 Spare Message French'
  510 = 'Clamp Cylinder A1 Failed to Advance... Check Q1.0...' | German: 'S1 510 Row 52 Failed To Advance.. Check Qxxx.x German' | French: 'S1 510 Row 52 Failed To Advance.. Check Qxxx.x French'
  511 = 'Clamp Cylinder A1 Failed to Return... Check Q1.1...' | German: 'S1 511 Row 52 Failed To Return.. Check Qxxx.x German' | French: 'S1 511 Row 52 Failed To Return.. Check Qxxx.x French'
  512 = 'Clamp Cylinder A1 Lost Advanced... Check I1.0...' | German: 'S1 512 Row 52 Lost Advance Position... Check Ixxx.x German' | French: 'S1 512 Row 52 Lost Advance Position... Check Ixxx.x French'
  513 = 'Clamp Cylinder A1 Lost Returned... Check I1.1...' | German: 'S1 513 Row 52 Lost Return Position... Check Ixxx.x German' | French: 'S1 513 Row 52 Lost Return Position... Check Ixxx.x French'
  514 = 'Clamp Cylinder A1 Switch Fault... Check I1.0, I1.1...' | German: 'S1 514 Row 52 Switch Fault... Check Ixxx.x / Ixxx.x German' | French: 'S1 514 Row 52 Switch Fault... Check Ixxx.x / Ixxx.x French'
  515 = 'Spare' | German: 'S1 515 Row 52 Spare Message German' | French: 'S1 515 Row 52 Spare Message French'
  516 = 'Spare' | German: 'S1 516 Row 52 Spare Message German' | French: 'S1 516 Row 52 Spare Message French'
  517 = 'Spare' | German: 'S1 517 Row 52 Spare Message German' | French: 'S1 517 Row 52 Spare Message French'
  518 = 'Spare' | German: 'S1 518 Row 52 Spare Message German' | French: 'S1 518 Row 52 Spare Message French'
  519 = 'Spare' | German: 'S1 519 Row 52 Spare Message German' | French: 'S1 519 Row 52 Spare Message French'
  520 = 'Clamp Cylinder A1 Failed to Advance... Check Q1.0...' | German: 'S1 520 Row 53 Failed To Advance.. Check Qxxx.x German' | French: 'S1 520 Row 53 Failed To Advance.. Check Qxxx.x French'
  521 = 'Clamp Cylinder A1 Failed to Return... Check Q1.1...' | German: 'S1 521 Row 53 Failed To Return.. Check Qxxx.x German' | French: 'S1 521 Row 53 Failed To Return.. Check Qxxx.x French'
  522 = 'Clamp Cylinder A1 Lost Advanced... Check I1.0...' | German: 'S1 522 Row 53 Lost Advance Position... Check Ixxx.x German' | French: 'S1 522 Row 53 Lost Advance Position... Check Ixxx.x French'
  523 = 'Clamp Cylinder A1 Lost Returned... Check I1.1...' | German: 'S1 523 Row 53 Lost Return Position... Check Ixxx.x German' | French: 'S1 523 Row 53 Lost Return Position... Check Ixxx.x French'
  524 = 'Clamp Cylinder A1 Switch Fault... Check I1.0, I1.1...' | German: 'S1 524 Row 53 Switch Fault... Check Ixxx.x / Ixxx.x German' | French: 'S1 524 Row 53 Switch Fault... Check Ixxx.x / Ixxx.x French'
  525 = 'Spare' | German: 'S1 525 Row 53 Spare Message German' | French: 'S1 525 Row 53 Spare Message French'
  526 = 'Spare' | German: 'S1 526 Row 53 Spare Message German' | French: 'S1 526 Row 53 Spare Message French'
  527 = 'Spare' | German: 'S1 527 Row 53 Spare Message German' | French: 'S1 527 Row 53 Spare Message French'
  528 = 'Spare' | German: 'S1 528 Row 53 Spare Message German' | French: 'S1 528 Row 53 Spare Message French'
  529 = 'Spare' | German: 'S1 529 Row 53 Spare Message German' | French: 'S1 529 Row 53 Spare Message French'
  530 = 'Clamp Cylinder A1 Failed to Advance... Check Q1.0...' | German: 'S1 530 Row 54 Failed To Advance.. Check Qxxx.x German' | French: 'S1 530 Row 54 Failed To Advance.. Check Qxxx.x French'
  531 = 'Clamp Cylinder A1 Failed to Return... Check Q1.1...' | German: 'S1 531 Row 54 Failed To Return.. Check Qxxx.x German' | French: 'S1 531 Row 54 Failed To Return.. Check Qxxx.x French'
  532 = 'Clamp Cylinder A1 Lost Advanced... Check I1.0...' | German: 'S1 532 Row 54 Lost Advance Position... Check Ixxx.x German' | French: 'S1 532 Row 54 Lost Advance Position... Check Ixxx.x French'
  533 = 'Clamp Cylinder A1 Lost Returned... Check I1.1...' | German: 'S1 533 Row 54 Lost Return Position... Check Ixxx.x German' | French: 'S1 533 Row 54 Lost Return Position... Check Ixxx.x French'
  534 = 'Clamp Cylinder A1 Switch Fault... Check I1.0, I1.1...' | German: 'S1 534 Row 54 Switch Fault... Check Ixxx.x / Ixxx.x German' | French: 'S1 534 Row 54 Switch Fault... Check Ixxx.x / Ixxx.x French'
  535 = 'Spare' | German: 'S1 535 Row 54 Spare Message German' | French: 'S1 535 Row 54 Spare Message French'
  536 = 'Spare' | German: 'S1 536 Row 54 Spare Message German' | French: 'S1 536 Row 54 Spare Message French'
  537 = 'Spare' | German: 'S1 537 Row 54 Spare Message German' | French: 'S1 537 Row 54 Spare Message French'
  538 = 'Spare' | German: 'S1 538 Row 54 Spare Message German' | French: 'S1 538 Row 54 Spare Message French'
  539 = 'Spare' | German: 'S1 539 Row 54 Spare Message German' | French: 'S1 539 Row 54 Spare Message French'
  540 = 'Clamp Cylinder A1 Failed to Advance... Check Q1.0...' | German: 'S1 540 Row 55 Failed To Advance.. Check Qxxx.x German' | French: 'S1 540 Row 55 Failed To Advance.. Check Qxxx.x French'
  541 = 'Clamp Cylinder A1 Failed to Return... Check Q1.1...' | German: 'S1 541 Row 55 Failed To Return.. Check Qxxx.x German' | French: 'S1 541 Row 55 Failed To Return.. Check Qxxx.x French'
  542 = 'Clamp Cylinder A1 Lost Advanced... Check I1.0...' | German: 'S1 542 Row 55 Lost Advance Position... Check Ixxx.x German' | French: 'S1 542 Row 55 Lost Advance Position... Check Ixxx.x French'
  543 = 'Clamp Cylinder A1 Lost Returned... Check I1.1...' | German: 'S1 543 Row 55 Lost Return Position... Check Ixxx.x German' | French: 'S1 543 Row 55 Lost Return Position... Check Ixxx.x French'
  544 = 'Clamp Cylinder A1 Switch Fault... Check I1.0, I1.1...' | German: 'S1 544 Row 55 Switch Fault... Check Ixxx.x / Ixxx.x German' | French: 'S1 544 Row 55 Switch Fault... Check Ixxx.x / Ixxx.x French'
  545 = 'Spare' | German: 'S1 545 Row 55 Spare Message German' | French: 'S1 545 Row 55 Spare Message French'
  546 = 'Spare' | German: 'S1 546 Row 55 Spare Message German' | French: 'S1 546 Row 55 Spare Message French'
  547 = 'Spare' | German: 'S1 547 Row 55 Spare Message German' | French: 'S1 547 Row 55 Spare Message French'
  548 = 'Spare' | German: 'S1 548 Row 55 Spare Message German' | French: 'S1 548 Row 55 Spare Message French'
  549 = 'Spare' | German: 'S1 549 Row 55 Spare Message German' | French: 'S1 549 Row 55 Spare Message French'
  550 = 'Clamp Cylinder A1 Failed to Advance... Check Q1.0...' | German: 'S1 550 Row 56 Failed To Advance.. Check Qxxx.x German' | French: 'S1 550 Row 56 Failed To Advance.. Check Qxxx.x French'
  551 = 'Clamp Cylinder A1 Failed to Return... Check Q1.1...' | German: 'S1 551 Row 56 Failed To Return.. Check Qxxx.x German' | French: 'S1 551 Row 56 Failed To Return.. Check Qxxx.x French'
  552 = 'Clamp Cylinder A1 Lost Advanced... Check I1.0...' | German: 'S1 552 Row 56 Lost Advance Position... Check Ixxx.x German' | French: 'S1 552 Row 56 Lost Advance Position... Check Ixxx.x French'
  553 = 'Clamp Cylinder A1 Lost Returned... Check I1.1...' | German: 'S1 553 Row 56 Lost Return Position... Check Ixxx.x German' | French: 'S1 553 Row 56 Lost Return Position... Check Ixxx.x French'
  554 = 'Clamp Cylinder A1 Switch Fault... Check I1.0, I1.1...' | German: 'S1 554 Row 56 Switch Fault... Check Ixxx.x / Ixxx.x German' | French: 'S1 554 Row 56 Switch Fault... Check Ixxx.x / Ixxx.x French'
  555 = 'Spare' | German: 'S1 555 Row 56 Spare Message German' | French: 'S1 555 Row 56 Spare Message French'
  556 = 'Spare' | German: 'S1 556 Row 56 Spare Message German' | French: 'S1 556 Row 56 Spare Message French'
  557 = 'Spare' | German: 'S1 557 Row 56 Spare Message German' | French: 'S1 557 Row 56 Spare Message French'
  558 = 'Spare' | German: 'S1 558 Row 56 Spare Message German' | French: 'S1 558 Row 56 Spare Message French'
  559 = 'Spare' | German: 'S1 559 Row 56 Spare Message German' | French: 'S1 559 Row 56 Spare Message French'
  560 = 'Clamp Cylinder A1 Failed to Advance... Check Q1.0...' | German: 'S1 560 Row 57 Failed To Advance.. Check Qxxx.x German' | French: 'S1 560 Row 57 Failed To Advance.. Check Qxxx.x French'
  561 = 'Clamp Cylinder A1 Failed to Return... Check Q1.1...' | German: 'S1 561 Row 57 Failed To Return.. Check Qxxx.x German' | French: 'S1 561 Row 57 Failed To Return.. Check Qxxx.x French'
  562 = 'Clamp Cylinder A1 Lost Advanced... Check I1.0...' | German: 'S1 562 Row 57 Lost Advance Position... Check Ixxx.x German' | French: 'S1 562 Row 57 Lost Advance Position... Check Ixxx.x French'
  563 = 'Clamp Cylinder A1 Lost Returned... Check I1.1...' | German: 'S1 563 Row 57 Lost Return Position... Check Ixxx.x German' | French: 'S1 563 Row 57 Lost Return Position... Check Ixxx.x French'
  564 = 'Clamp Cylinder A1 Switch Fault... Check I1.0, I1.1...' | German: 'S1 564 Row 57 Switch Fault... Check Ixxx.x / Ixxx.x German' | French: 'S1 564 Row 57 Switch Fault... Check Ixxx.x / Ixxx.x French'
  565 = 'Spare' | German: 'S1 565 Row 57 Spare Message German' | French: 'S1 565 Row 57 Spare Message French'
  566 = 'Spare' | German: 'S1 566 Row 57 Spare Message German' | French: 'S1 566 Row 57 Spare Message French'
  567 = 'Spare' | German: 'S1 567 Row 57 Spare Message German' | French: 'S1 567 Row 57 Spare Message French'
  568 = 'Spare' | German: 'S1 568 Row 57 Spare Message German' | French: 'S1 568 Row 57 Spare Message French'
  569 = 'Spare' | German: 'S1 569 Row 57 Spare Message German' | French: 'S1 569 Row 57 Spare Message French'
  570 = 'Clamp Cylinder A1 Failed to Advance... Check Q1.0...' | German: 'S1 570 Row 58 Failed To Advance.. Check Qxxx.x German' | French: 'S1 570 Row 58 Failed To Advance.. Check Qxxx.x French'
  571 = 'Clamp Cylinder A1 Failed to Return... Check Q1.1...' | German: 'S1 571 Row 58 Failed To Return.. Check Qxxx.x German' | French: 'S1 571 Row 58 Failed To Return.. Check Qxxx.x French'
  572 = 'Clamp Cylinder A1 Lost Advanced... Check I1.0...' | German: 'S1 572 Row 58 Lost Advance Position... Check Ixxx.x German' | French: 'S1 572 Row 58 Lost Advance Position... Check Ixxx.x French'
  573 = 'Clamp Cylinder A1 Lost Returned... Check I1.1...' | German: 'S1 573 Row 58 Lost Return Position... Check Ixxx.x German' | French: 'S1 573 Row 58 Lost Return Position... Check Ixxx.x French'
  574 = 'Clamp Cylinder A1 Switch Fault... Check I1.0, I1.1...' | German: 'S1 574 Row 58 Switch Fault... Check Ixxx.x / Ixxx.x German' | French: 'S1 574 Row 58 Switch Fault... Check Ixxx.x / Ixxx.x French'
  575 = 'Spare' | German: 'S1 575 Row 58 Spare Message German' | French: 'S1 575 Row 58 Spare Message French'
  576 = 'Spare' | German: 'S1 576 Row 58 Spare Message German' | French: 'S1 576 Row 58 Spare Message French'
  577 = 'Spare' | German: 'S1 577 Row 58 Spare Message German' | French: 'S1 577 Row 58 Spare Message French'
  578 = 'Spare' | German: 'S1 578 Row 58 Spare Message German' | French: 'S1 578 Row 58 Spare Message French'
  579 = 'Spare' | German: 'S1 579 Row 58 Spare Message German' | French: 'S1 579 Row 58 Spare Message French'
  580 = 'Clamp Cylinder A1 Failed to Advance... Check Q1.0...' | German: 'S1 580 Row 59 Failed To Advance.. Check Qxxx.x German' | French: 'S1 580 Row 59 Failed To Advance.. Check Qxxx.x French'
  581 = 'Clamp Cylinder A1 Failed to Return... Check Q1.1...' | German: 'S1 581 Row 59 Failed To Return.. Check Qxxx.x German' | French: 'S1 581 Row 59 Failed To Return.. Check Qxxx.x French'
  582 = 'Clamp Cylinder A1 Lost Advanced... Check I1.0...' | German: 'S1 582 Row 59 Lost Advance Position... Check Ixxx.x German' | French: 'S1 582 Row 59 Lost Advance Position... Check Ixxx.x French'
  583 = 'Clamp Cylinder A1 Lost Returned... Check I1.1...' | German: 'S1 583 Row 59 Lost Return Position... Check Ixxx.x German' | French: 'S1 583 Row 59 Lost Return Position... Check Ixxx.x French'
  584 = 'Clamp Cylinder A1 Switch Fault... Check I1.0, I1.1...' | German: 'S1 584 Row 59 Switch Fault... Check Ixxx.x / Ixxx.x German' | French: 'S1 584 Row 59 Switch Fault... Check Ixxx.x / Ixxx.x French'
  585 = 'Spare' | German: 'S1 585 Row 59 Spare Message German' | French: 'S1 585 Row 59 Spare Message French'
  586 = 'Spare' | German: 'S1 586 Row 59 Spare Message German' | French: 'S1 586 Row 59 Spare Message French'
  587 = 'Spare' | German: 'S1 587 Row 59 Spare Message German' | French: 'S1 587 Row 59 Spare Message French'
  588 = 'Spare' | German: 'S1 588 Row 59 Spare Message German' | French: 'S1 588 Row 59 Spare Message French'
  589 = 'Spare' | German: 'S1 589 Row 59 Spare Message German' | French: 'S1 589 Row 59 Spare Message French'
  590 = 'Clamp Cylinder A1 Failed to Advance... Check Q1.0...' | German: 'S1 590 Row 60 Failed To Advance.. Check Qxxx.x German' | French: 'S1 590 Row 60 Failed To Advance.. Check Qxxx.x French'
  591 = 'Clamp Cylinder A1 Failed to Return... Check Q1.1...' | German: 'S1 591 Row 60 Failed To Return.. Check Qxxx.x German' | French: 'S1 591 Row 60 Failed To Return.. Check Qxxx.x French'
  592 = 'Clamp Cylinder A1 Lost Advanced... Check I1.0...' | German: 'S1 592 Row 60 Lost Advance Position... Check Ixxx.x German' | French: 'S1 592 Row 60 Lost Advance Position... Check Ixxx.x French'
  593 = 'Clamp Cylinder A1 Lost Returned... Check I1.1...' | German: 'S1 593 Row 60 Lost Return Position... Check Ixxx.x German' | French: 'S1 593 Row 60 Lost Return Position... Check Ixxx.x French'
  594 = 'Clamp Cylinder A1 Switch Fault... Check I1.0, I1.1...' | German: 'S1 594 Row 60 Switch Fault... Check Ixxx.x / Ixxx.x German' | French: 'S1 594 Row 60 Switch Fault... Check Ixxx.x / Ixxx.x French'
  595 = 'Spare' | German: 'S1 595 Row 60 Spare Message German' | French: 'S1 595 Row 60 Spare Message French'
  596 = 'Spare' | German: 'S1 596 Row 60 Spare Message German' | French: 'S1 596 Row 60 Spare Message French'
  597 = 'Spare' | German: 'S1 597 Row 60 Spare Message German' | French: 'S1 597 Row 60 Spare Message French'
  598 = 'Spare' | German: 'S1 598 Row 60 Spare Message German' | French: 'S1 598 Row 60 Spare Message French'
  599 = 'Spare' | German: 'S1 599 Row 60 Spare Message German' | French: 'S1 599 Row 60 Spare Message French'
  600 = 'Clamp Cylinder A1 Failed to Advance... Check Q1.0...' | German: 'S1 600 Row 61 Failed To Advance.. Check Qxxx.x German' | French: 'S1 600 Row 61 Failed To Advance.. Check Qxxx.x French'
  601 = 'Clamp Cylinder A1 Failed to Return... Check Q1.1...' | German: 'S1 601 Row 61 Failed To Return.. Check Qxxx.x German' | French: 'S1 601 Row 61 Failed To Return.. Check Qxxx.x French'
  602 = 'Clamp Cylinder A1 Lost Advanced... Check I1.0...' | German: 'S1 602 Row 61 Lost Advance Position... Check Ixxx.x German' | French: 'S1 602 Row 61 Lost Advance Position... Check Ixxx.x French'
  603 = 'Clamp Cylinder A1 Lost Returned... Check I1.1...' | German: 'S1 603 Row 61 Lost Return Position... Check Ixxx.x German' | French: 'S1 603 Row 61 Lost Return Position... Check Ixxx.x French'
  604 = 'Clamp Cylinder A1 Switch Fault... Check I1.0, I1.1...' | German: 'S1 604 Row 61 Switch Fault... Check Ixxx.x / Ixxx.x German' | French: 'S1 604 Row 61 Switch Fault... Check Ixxx.x / Ixxx.x French'
  605 = 'Spare' | German: 'S1 605 Row 61 Spare Message German' | French: 'S1 605 Row 61 Spare Message French'
  606 = 'Spare' | German: 'S1 606 Row 61 Spare Message German' | French: 'S1 606 Row 61 Spare Message French'
  607 = 'Spare' | German: 'S1 607 Row 61 Spare Message German' | French: 'S1 607 Row 61 Spare Message French'
  608 = 'Spare' | German: 'S1 608 Row 61 Spare Message German' | French: 'S1 608 Row 61 Spare Message French'
  609 = 'Spare' | German: 'S1 609 Row 61 Spare Message German' | French: 'S1 609 Row 61 Spare Message French'
  610 = 'Clamp Cylinder A1 Failed to Advance... Check Q1.0...' | German: 'S1 610 Row 62 Failed To Advance.. Check Qxxx.x German' | French: 'S1 610 Row 62 Failed To Advance.. Check Qxxx.x French'
  611 = 'Clamp Cylinder A1 Failed to Return... Check Q1.1...' | German: 'S1 611 Row 62 Failed To Return.. Check Qxxx.x German' | French: 'S1 611 Row 62 Failed To Return.. Check Qxxx.x French'
  612 = 'Clamp Cylinder A1 Lost Advanced... Check I1.0...' | German: 'S1 612 Row 62 Lost Advance Position... Check Ixxx.x German' | French: 'S1 612 Row 62 Lost Advance Position... Check Ixxx.x French'
  613 = 'Clamp Cylinder A1 Lost Returned... Check I1.1...' | German: 'S1 613 Row 62 Lost Return Position... Check Ixxx.x German' | French: 'S1 613 Row 62 Lost Return Position... Check Ixxx.x French'
  614 = 'Clamp Cylinder A1 Switch Fault... Check I1.0, I1.1...' | German: 'S1 614 Row 62 Switch Fault... Check Ixxx.x / Ixxx.x German' | French: 'S1 614 Row 62 Switch Fault... Check Ixxx.x / Ixxx.x French'
  615 = 'Spare' | German: 'S1 615 Row 62 Spare Message German' | French: 'S1 615 Row 62 Spare Message French'
  616 = 'Spare' | German: 'S1 616 Row 62 Spare Message German' | French: 'S1 616 Row 62 Spare Message French'
  617 = 'Spare' | German: 'S1 617 Row 62 Spare Message German' | French: 'S1 617 Row 62 Spare Message French'
  618 = 'Spare' | German: 'S1 618 Row 62 Spare Message German' | French: 'S1 618 Row 62 Spare Message French'
  619 = 'Spare' | German: 'S1 619 Row 62 Spare Message German' | French: 'S1 619 Row 62 Spare Message French'
  620 = 'Clamp Cylinder A1 Failed to Advance... Check Q1.0...' | German: 'S1 620 Row 63 Failed To Advance.. Check Qxxx.x German' | French: 'S1 620 Row 63 Failed To Advance.. Check Qxxx.x French'
  621 = 'Clamp Cylinder A1 Failed to Return... Check Q1.1...' | German: 'S1 621 Row 63 Failed To Return.. Check Qxxx.x German' | French: 'S1 621 Row 63 Failed To Return.. Check Qxxx.x French'
  622 = 'Clamp Cylinder A1 Lost Advanced... Check I1.0...' | German: 'S1 622 Row 63 Lost Advance Position... Check Ixxx.x German' | French: 'S1 622 Row 63 Lost Advance Position... Check Ixxx.x French'
  623 = 'Clamp Cylinder A1 Lost Returned... Check I1.1...' | German: 'S1 623 Row 63 Lost Return Position... Check Ixxx.x German' | French: 'S1 623 Row 63 Lost Return Position... Check Ixxx.x French'
  624 = 'Clamp Cylinder A1 Switch Fault... Check I1.0, I1.1...' | German: 'S1 624 Row 63 Switch Fault... Check Ixxx.x / Ixxx.x German' | French: 'S1 624 Row 63 Switch Fault... Check Ixxx.x / Ixxx.x French'
  625 = 'Spare' | German: 'S1 625 Row 63 Spare Message German' | French: 'S1 625 Row 63 Spare Message French'
  626 = 'Spare' | German: 'S1 626 Row 63 Spare Message German' | French: 'S1 626 Row 63 Spare Message French'
  627 = 'Spare' | German: 'S1 627 Row 63 Spare Message German' | French: 'S1 627 Row 63 Spare Message French'
  628 = 'Spare' | German: 'S1 628 Row 63 Spare Message German' | French: 'S1 628 Row 63 Spare Message French'
  629 = 'Spare' | German: 'S1 629 Row 63 Spare Message German' | French: 'S1 629 Row 63 Spare Message French'
  630 = 'Clamp Cylinder A1 Failed to Advance... Check Q1.0...' | German: 'S1 630 Row 64 Failed To Advance.. Check Qxxx.x German' | French: 'S1 630 Row 64 Failed To Advance.. Check Qxxx.x French'
  631 = 'Clamp Cylinder A1 Failed to Return... Check Q1.1...' | German: 'S1 631 Row 64 Failed To Return.. Check Qxxx.x German' | French: 'S1 631 Row 64 Failed To Return.. Check Qxxx.x French'
  632 = 'Clamp Cylinder A1 Lost Advanced... Check I1.0...' | German: 'S1 632 Row 64 Lost Advance Position... Check Ixxx.x German' | French: 'S1 632 Row 64 Lost Advance Position... Check Ixxx.x French'
  633 = 'Clamp Cylinder A1 Lost Returned... Check I1.1...' | German: 'S1 633 Row 64 Lost Return Position... Check Ixxx.x German' | French: 'S1 633 Row 64 Lost Return Position... Check Ixxx.x French'
  634 = 'Clamp Cylinder A1 Switch Fault... Check I1.0, I1.1...' | German: 'S1 634 Row 64 Switch Fault... Check Ixxx.x / Ixxx.x German' | French: 'S1 634 Row 64 Switch Fault... Check Ixxx.x / Ixxx.x French'
  635 = 'Spare' | German: 'S1 635 Row 64 Spare Message German' | French: 'S1 635 Row 64 Spare Message French'
  636 = 'Spare' | German: 'S1 636 Row 64 Spare Message German' | French: 'S1 636 Row 64 Spare Message French'
  637 = 'Spare' | German: 'S1 637 Row 64 Spare Message German' | French: 'S1 637 Row 64 Spare Message French'
  638 = 'Spare' | German: 'S1 638 Row 64 Spare Message German' | French: 'S1 638 Row 64 Spare Message French'
  639 = 'Spare' | German: 'S1 639 Row 64 Spare Message German' | French: 'S1 639 Row 64 Spare Message French'
  640 = 'Clamp Cylinder A1 Failed to Advance... Check Q1.0...' | German: 'S1 640 Row 65 Failed To Advance.. Check Qxxx.x German' | French: 'S1 640 Row 65 Failed To Advance.. Check Qxxx.x French'
  641 = 'Clamp Cylinder A1 Failed to Return... Check Q1.1...' | German: 'S1 641 Row 65 Failed To Return.. Check Qxxx.x German' | French: 'S1 641 Row 65 Failed To Return.. Check Qxxx.x French'
  642 = 'Clamp Cylinder A1 Lost Advanced... Check I1.0...' | German: 'S1 642 Row 65 Lost Advance Position... Check Ixxx.x German' | French: 'S1 642 Row 65 Lost Advance Position... Check Ixxx.x French'
  643 = 'Clamp Cylinder A1 Lost Returned... Check I1.1...' | German: 'S1 643 Row 65 Lost Return Position... Check Ixxx.x German' | French: 'S1 643 Row 65 Lost Return Position... Check Ixxx.x French'
  644 = 'Clamp Cylinder A1 Switch Fault... Check I1.0, I1.1...' | German: 'S1 644 Row 65 Switch Fault... Check Ixxx.x / Ixxx.x German' | French: 'S1 644 Row 65 Switch Fault... Check Ixxx.x / Ixxx.x French'
  645 = 'Spare' | German: 'S1 645 Row 65 Spare Message German' | French: 'S1 645 Row 65 Spare Message French'
  646 = 'Spare' | German: 'S1 646 Row 65 Spare Message German' | French: 'S1 646 Row 65 Spare Message French'
  647 = 'Spare' | German: 'S1 647 Row 65 Spare Message German' | French: 'S1 647 Row 65 Spare Message French'
  648 = 'Spare' | German: 'S1 648 Row 65 Spare Message German' | French: 'S1 648 Row 65 Spare Message French'
  649 = 'Spare' | German: 'S1 649 Row 65 Spare Message German' | French: 'S1 649 Row 65 Spare Message French'
